KUKA KRL program: MyProgram_114().src

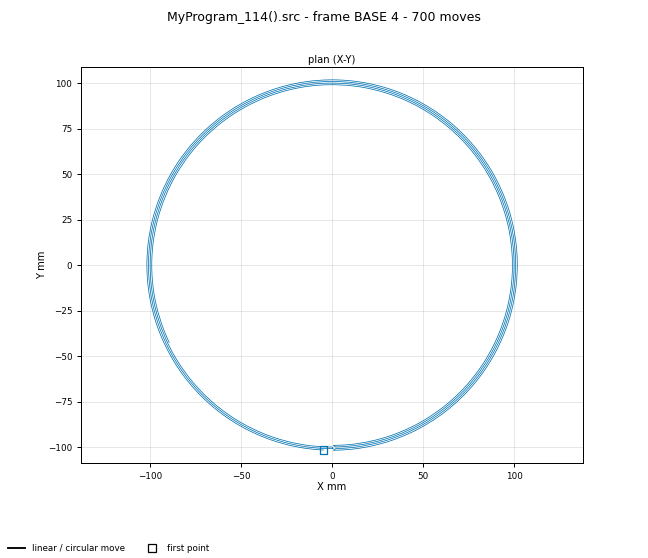
[picture p0: tool path of MyProgram_114().src in frame BASE 4, 700 of 700 moves have a stored position in this frame; points joined in program order, loops and branches not executed]
&ACCESS RVP
&REL 1
&PARAM TEMPLATE = C:\KRC\Roboter\Template\vorgabe
&PARAM EDITMASK = *
DEF MyProgram_114()
; ---- Setting reference (Base) ----
$BASE = BASE_DATA[4]

; --------------------------
; ---- Setting tool (TCP) ----
$TOOL = TOOL_DATA[3]
; --------------------------

$VEL.CP = VEL_APROX_PRINT
Startdeposition()
$VEL.CP = VEL_PRINT
LIN {X -4.7192,Y -101.6599,Z 99,A -97.1111,B 24.9445,C -1.7205,E1 24.9918,E2 182.675} C_DIS
LIN {X -7.4867,Y -101.4949,Z 99,A -98.6462,B 24.9445,C -1.7214,E1 24.9876,E2 184.2085} C_DIS
LIN {X -9.7017,Y -101.3059,Z 99,A -99.8982,B 24.9445,C -1.7214,E1 24.9841,E2 185.4609} C_DIS
LIN {X -12.4578,Y -101.0053,Z 99,A -101.4595,B 24.9445,C -1.7217,E1 24.9798,E2 187.0228} C_DIS
LIN {X -14.6609,Y -100.7078,Z 99,A -102.7373,B 24.9445,C -1.721,E1 24.9762,E2 188.3032} C_DIS
LIN {X -17.1279,Y -100.3177,Z 99,A -104.1189,B 24.9445,C -1.7223,E1 24.9724,E2 189.6829} C_DIS
LIN {X -19.8545,Y -99.8152,Z 99,A -105.6809,B 24.9444,C -1.7228,E1 24.9681,E2 191.2454} C_DIS
LIN {X -22.0297,Y -99.3564,Z 99,A -106.9595,B 24.9444,C -1.7224,E1 24.9646,E2 192.5265} C_DIS
LIN {X -24.4614,Y -98.7858,Z 99,A -108.3414,B 24.9443,C -1.7241,E1 24.9609,E2 193.9064} C_DIS
LIN {X -27.1435,Y -98.0841,Z 99,A -109.9045,B 24.9443,C -1.7249,E1 24.9567,E2 195.4699} C_DIS
LIN {X -29.2791,Y -97.4666,Z 99,A -111.184,B 24.9443,C -1.7248,E1 24.9532,E2 196.7519} C_DIS
LIN {X -31.5189,Y -96.7651,Z 99,A -112.5378,B 24.9443,C -1.7246,E1 24.9496,E2 198.1085} C_DIS
LIN {X -34.2855,Y -95.8216,Z 99,A -114.1306,B 24.944,C -1.7279,E1 24.9454,E2 199.6966} C_DIS
LIN {X -36.6268,Y -94.9513,Z 99,A -115.5395,B 24.944,C -1.7291,E1 24.9418,E2 201.1056} C_DIS
LIN {X -38.6915,Y -94.1274,Z 99,A -116.7915,B 24.9439,C -1.7303,E1 24.9385,E2 202.3574} C_DIS
LIN {X -40.9898,Y -93.1495,Z 99,A -118.2034,B 24.9439,C -1.7316,E1 24.9349,E2 203.7695} C_DIS
LIN {X -43.5126,Y -91.9996,Z 99,A -119.7683,B 24.9437,C -1.7333,E1 24.9309,E2 205.3344} C_DIS
LIN {X -45.5111,Y -91.026,Z 99,A -121.0488,B 24.9437,C -1.7338,E1 24.9277,E2 206.6171} C_DIS
LIN {X -48.4255,Y -89.509,Z 99,A -122.9613,B 24.9437,C -1.7339,E1 24.923,E2 208.5346} C_DIS
LIN {X -51.2454,Y -87.9271,Z 99,A -124.7043,B 24.9433,C -1.7392,E1 24.9188,E2 210.2701} C_DIS
LIN {X -53.1531,Y -86.7857,Z 99,A -125.9857,B 24.9433,C -1.74,E1 24.9157,E2 211.5535} C_DIS
LIN {X -55.4981,Y -85.3067,Z 99,A -127.5259,B 24.9431,C -1.7431,E1 24.9121,E2 213.0913} C_DIS
LIN {X -57.5749,Y -83.919,Z 99,A -128.9373,B 24.9429,C -1.7452,E1 24.9088,E2 214.5024} C_DIS
LIN {X -60.0996,Y -82.1274,Z 99,A -130.7649,B 24.9429,C -1.7452,E1 24.9047,E2 216.3365} C_DIS
LIN {X -62.3949,Y -80.3982,Z 99,A -132.3189,B 24.9426,C -1.7503,E1 24.9012,E2 217.8839} C_DIS
LIN {X -64.3492,Y -78.8428,Z 99,A -133.7487,B 24.9425,C -1.7521,E1 24.8981,E2 219.3149} C_DIS
LIN {X -66.4738,Y -77.0616,Z 99,A -135.2899,B 24.9422,C -1.7557,E1 24.8949,E2 220.8533} C_DIS
LIN {X -68.345,Y -75.4071,Z 99,A -136.7026,B 24.9421,C -1.7583,E1 24.8919,E2 222.2655} C_DIS
LIN {X -70.8764,Y -73.031,Z 99,A -138.666,B 24.9418,C -1.762,E1 24.8879,E2 224.2282} C_DIS
LIN {X -72.8404,Y -71.0742,Z 99,A -140.2343,B 24.9416,C -1.7651,E1 24.8849,E2 225.7959} C_DIS
LIN {X -74.5627,Y -69.2652,Z 99,A -141.6473,B 24.9414,C -1.7679,E1 24.8822,E2 227.2083} C_DIS
LIN {X -76.0569,Y -67.6192,Z 99,A -142.9199,B 24.9413,C -1.77,E1 24.8798,E2 228.4816} C_DIS
LIN {X -77.6934,Y -65.7323,Z 99,A -144.3182,B 24.941,C -1.7735,E1 24.8772,E2 229.8779} C_DIS
LIN {X -79.4561,Y -63.5924,Z 99,A -145.8873,B 24.9408,C -1.7769,E1 24.8745,E2 231.4463} C_DIS
LIN {X -80.9928,Y -61.6233,Z 99,A -147.3008,B 24.9406,C -1.78,E1 24.8721,E2 232.859} C_DIS
LIN {X -83.2061,Y -58.6004,Z 99,A -149.4215,B 24.9403,C -1.7848,E1 24.8686,E2 234.9785} C_DIS
LIN {X -85.1119,Y -55.7934,Z 99,A -151.3537,B 24.94,C -1.789,E1 24.8656,E2 236.9105} C_DIS
LIN {X -86.4974,Y -53.6208,Z 99,A -152.8276,B 24.9398,C -1.7919,E1 24.8634,E2 238.3848} C_DIS
LIN {X -87.9271,Y -51.2454,Z 99,A -154.3716,B 24.9395,C -1.7966,E1 24.8612,E2 239.9256} C_DIS
LIN {X -89.1582,Y -49.0722,Z 99,A -155.7862,B 24.9393,C -1.8002,E1 24.8593,E2 241.3392} C_DIS
LIN {X -90.2077,Y -47.1124,Z 99,A -157.0452,B 24.939,C -1.8033,E1 24.8576,E2 242.5974} C_DIS
LIN {X -91.4587,Y -44.6383,Z 99,A -158.6156,B 24.9388,C -1.8073,E1 24.8557,E2 244.1667} C_DIS
LIN {X -92.4107,Y -42.6294,Z 99,A -159.9009,B 24.9386,C -1.8097,E1 24.8542,E2 245.4533} C_DIS
LIN {X -93.5388,Y -40.0968,Z 99,A -161.4454,B 24.9383,C -1.8147,E1 24.8524,E2 246.9944} C_DIS
LIN {X -94.4947,Y -37.7892,Z 99,A -162.8609,B 24.938,C -1.8185,E1 24.8509,E2 248.4088} C_DIS
LIN {X -95.6293,Y -34.8126,Z 99,A -164.7206,B 24.9378,C -1.8215,E1 24.8491,E2 250.2717} C_DIS
LIN {X -96.5463,Y -32.1839,Z 99,A -166.2697,B 24.9374,C -1.8268,E1 24.8477,E2 251.817} C_DIS
LIN {X -97.3071,Y -29.8049,Z 99,A -167.6851,B 24.9372,C -1.8307,E1 24.8465,E2 253.2313} C_DIS
LIN {X -98.0787,Y -27.1626,Z 99,A -169.2166,B 24.9368,C -1.836,E1 24.8454,E2 254.759} C_DIS
LIN {X -98.7207,Y -24.7283,Z 99,A -170.6462,B 24.9365,C -1.8399,E1 24.8444,E2 256.1876} C_DIS
LIN {X -99.236,Y -22.5657,Z 99,A -171.932,B 24.9364,C -1.8426,E1 24.8436,E2 257.4745} C_DIS
LIN {X -99.7649,Y -20.0991,Z 99,A -173.3334,B 24.936,C -1.8477,E1 24.8428,E2 258.8721} C_DIS
LIN {X -100.1715,Y -17.9594,Z 99,A -174.6638,B 24.936,C -1.848,E1 24.8421,E2 260.2096} C_DIS
LIN {X -100.6272,Y -15.2044,Z 99,A -176.1799,B 24.9355,C -1.8548,E1 24.8414,E2 261.7185} C_DIS
LIN {X -100.97,Y -12.7303,Z 99,A -177.5957,B 24.9352,C -1.859,E1 24.8409,E2 263.1329} C_DIS
LIN {X -101.3347,Y -9.3895,Z 99,A -179.5206,B 24.9349,C -1.8639,E1 24.8404,E2 265.0576} C_DIS
LIN {X -101.5606,Y -6.5147,Z 99,A 178.89,B 24.9344,C -1.8702,E1 24.8401,E2 266.6414} C_DIS
LIN {X -101.7017,Y -3.7459,Z 99,A 177.3182,B 24.9341,C -1.8748,E1 24.8399,E2 268.2118} C_DIS
LIN {X -101.763,Y -1.2489,Z 99,A 175.8879,B 24.9338,C -1.8785,E1 24.8398,E2 269.6418} C_DIS
LIN {X -101.763,Y 1.2489,Z 99,A 174.2862,B 24.934,C -1.8764,E1 24.8398,E2 271.2582} C_DIS
LIN {X -101.6599,Y 4.7192,Z 99,A 172.4912,B 24.9332,C -1.8881,E1 24.84,E2 273.036} C_DIS
LIN {X -101.4949,Y 7.4867,Z 99,A 170.9451,B 24.9328,C -1.8936,E1 24.8403,E2 274.5783} C_DIS
LIN {X -101.3059,Y 9.7017,Z 99,A 169.6846,B 24.9325,C -1.8974,E1 24.8406,E2 275.8374} C_DIS
LIN {X -101.0053,Y 12.4578,Z 99,A 168.1128,B 24.9322,C -1.902,E1 24.8411,E2 277.4075} C_DIS
LIN {X -100.4783,Y 16.1671,Z 99,A 165.9887,B 24.9317,C -1.9083,E1 24.842,E2 279.5293} C_DIS
LIN {X -100.0513,Y 18.6281,Z 99,A 164.5726,B 24.9314,C -1.9125,E1 24.8427,E2 280.9438} C_DIS
LIN {X -99.6192,Y 20.8088,Z 99,A 163.2861,B 24.9312,C -1.9153,E1 24.8434,E2 282.2312} C_DIS
LIN {X -99.0786,Y 23.2473,Z 99,A 161.8959,B 24.9309,C -1.9203,E1 24.8443,E2 283.6176} C_DIS
LIN {X -98.4098,Y 25.9378,Z 99,A 160.3241,B 24.9305,C -1.9249,E1 24.8453,E2 285.1877} C_DIS
LIN {X -97.7436,Y 28.3451,Z 99,A 158.9084,B 24.9302,C -1.929,E1 24.8464,E2 286.6018} C_DIS
LIN {X -97.0186,Y 30.7353,Z 99,A 157.4927,B 24.9299,C -1.9331,E1 24.8476,E2 288.016} C_DIS
LIN {X -96.3229,Y 32.8467,Z 99,A 156.2321,B 24.9297,C -1.9367,E1 24.8487,E2 289.2751} C_DIS
LIN {X -95.5717,Y 34.9704,Z 99,A 154.8757,B 24.9297,C -1.9376,E1 24.85,E2 290.637} C_DIS
LIN {X -94.4947,Y 37.7892,Z 99,A 153.2451,B 24.9291,C -1.9451,E1 24.8516,E2 292.2587} C_DIS
LIN {X -93.6455,Y 39.8437,Z 99,A 151.9848,B 24.9288,C -1.9487,E1 24.853,E2 293.5177} C_DIS
LIN {X -92.6395,Y 42.1298,Z 99,A 150.5435,B 24.9286,C -1.9517,E1 24.8546,E2 294.9595} C_DIS
LIN {X -91.4587,Y 44.6383,Z 99,A 148.9981,B 24.9282,C -1.9569,E1 24.8565,E2 296.501} C_DIS
LIN {X -90.4607,Y 46.6247,Z 99,A 147.7128,B 24.928,C -1.9594,E1 24.8581,E2 297.7871} C_DIS
LIN {X -89.2892,Y 48.8307,Z 99,A 146.3231,B 24.9277,C -1.9641,E1 24.86,E2 299.173} C_DIS
LIN {X -87.9271,Y 51.2454,Z 99,A 144.6209,B 24.9277,C -1.9638,E1 24.8623,E2 300.8848} C_DIS
LIN {X -86.2717,Y 53.9822,Z 99,A 142.8532,B 24.9272,C -1.9701,E1 24.8649,E2 302.6466} C_DIS
LIN {X -84.7704,Y 56.3114,Z 99,A 141.3448,B 24.9268,C -1.9762,E1 24.8672,E2 304.148} C_DIS
LIN {X -83.363,Y 58.3748,Z 99,A 139.93,B 24.9265,C -1.9798,E1 24.8695,E2 305.5613} C_DIS
LIN {X -81.743,Y 60.6247,Z 99,A 138.3857,B 24.9262,C -1.9846,E1 24.872,E2 307.1017} C_DIS
LIN {X -80.2305,Y 62.6125,Z 99,A 136.9712,B 24.9259,C -1.988,E1 24.8744,E2 308.5145} C_DIS
LIN {X -78.8428,Y 64.3492,Z 99,A 135.7122,B 24.9257,C -1.9911,E1 24.8766,E2 309.7722} C_DIS
LIN {X -77.2398,Y 66.2647,Z 99,A 134.2982,B 24.9254,C -1.9945,E1 24.8792,E2 311.1846} C_DIS
LIN {X -75.4071,Y 68.345,Z 99,A 132.7287,B 24.9251,C -1.9981,E1 24.8821,E2 312.7524} C_DIS
LIN {X -73.7071,Y 70.175,Z 99,A 131.3148,B 24.9249,C -2.0013,E1 24.8848,E2 314.1649} C_DIS
LIN {X -71.9627,Y 71.9627,Z 99,A 129.901,B 24.9247,C -2.0045,E1 24.8875,E2 315.5771} C_DIS
LIN {X -70.175,Y 73.7071,Z 99,A 128.4875,B 24.9244,C -2.0076,E1 24.8904,E2 316.9892} C_DIS
LIN {X -68.5474,Y 75.2213,Z 99,A 127.2293,B 24.9242,C -2.0103,E1 24.893,E2 318.246} C_DIS
LIN {X -66.7956,Y 76.7806,Z 99,A 125.8457,B 24.9242,C -2.0111,E1 24.8959,E2 319.6332} C_DIS
LIN {X -64.7739,Y 78.4942,Z 99,A 124.3773,B 24.9239,C -2.0152,E1 24.899,E2 321.0975} C_DIS
LIN {X -62.8952,Y 80.0071,Z 99,A 122.9966,B 24.9237,C -2.0173,E1 24.902,E2 322.4781} C_DIS
LIN {X -60.6247,Y 81.743,Z 99,A 121.4223,B 24.9233,C -2.0219,E1 24.9055,E2 324.0472} C_DIS
LIN {X -58.6004,Y 83.2061,Z 99,A 120.0099,B 24.9231,C -2.0245,E1 24.9087,E2 325.4583} C_DIS
LIN {X -55.4981,Y 85.3067,Z 99,A 117.8912,B 24.9229,C -2.0283,E1 24.9137,E2 327.5749} C_DIS
LIN {X -53.6208,Y 86.4974,Z 99,A 116.6087,B 24.9228,C -2.0296,E1 24.9167,E2 328.8585} C_DIS
LIN {X -51.2454,Y 87.9271,Z 99,A 115.0673,B 24.9225,C -2.0331,E1 24.9204,E2 330.3962} C_DIS
LIN {X -49.312,Y 89.0243,Z 99,A 113.8175,B 24.9223,C -2.0353,E1 24.9234,E2 331.6443} C_DIS
LIN {X -47.1124,Y 90.2077,Z 99,A 112.3814,B 24.9223,C -2.0366,E1 24.927,E2 333.0813} C_DIS
LIN {X -44.6383,Y 91.4587,Z 99,A 110.8334,B 24.922,C -2.0396,E1 24.9308,E2 334.6264} C_DIS
LIN {X -42.3803,Y 92.5266,Z 99,A 109.4227,B 24.9218,C -2.0416,E1 24.9344,E2 336.0358} C_DIS
LIN {X -40.0968,Y 93.5388,Z 99,A 108.0119,B 24.9217,C -2.0435,E1 24.938,E2 337.4455} C_DIS
LIN {X -37.7892,Y 94.4947,Z 99,A 106.6008,B 24.9216,C -2.0453,E1 24.9417,E2 338.8555} C_DIS
LIN {X -35.7157,Y 95.2963,Z 99,A 105.3459,B 24.9214,C -2.0468,E1 24.9449,E2 340.1094} C_DIS
LIN {X -33.3663,Y 96.1441,Z 99,A 103.9356,B 24.9214,C -2.0485,E1 24.9486,E2 341.5186} C_DIS
LIN {X -30.7353,Y 97.0186,Z 99,A 102.371,B 24.9212,C -2.0502,E1 24.9528,E2 343.0819} C_DIS
LIN {X -27.7971,Y 97.8989,Z 99,A 100.5535,B 24.9212,C -2.0488,E1 24.9577,E2 344.9057} C_DIS
LIN {X -24.7283,Y 98.7207,Z 99,A 98.8471,B 24.9209,C -2.0535,E1 24.9623,E2 346.6034} C_DIS
LIN {X -21.2106,Y 99.5351,Z 99,A 96.8033,B 24.9209,C -2.055,E1 24.9678,E2 348.6464} C_DIS
LIN {X -18.8979,Y 99.9994,Z 99,A 95.4541,B 24.9208,C -2.0553,E1 24.9715,E2 349.9963} C_DIS
LIN {X -16.1671,Y 100.4783,Z 99,A 93.9164,B 24.9206,C -2.0572,E1 24.9757,E2 351.5309} C_DIS
LIN {X -12.7303,Y 100.97,Z 99,A 91.9591,B 24.9206,C -2.0584,E1 24.9812,E2 353.4869} C_DIS
LIN {X -9.9753,Y 101.2806,Z 99,A 90.3962,B 24.9205,C -2.0591,E1 24.9855,E2 355.0489} C_DIS
LIN {X -7.4867,Y 101.4949,Z 99,A 88.9887,B 24.9205,C -2.0597,E1 24.9894,E2 356.4557} C_DIS
LIN {X -5.2679,Y 101.6329,Z 99,A 87.7102,B 24.9205,C -2.0592,E1 24.993,E2 357.7357} C_DIS
LIN {X -1.6701,Y 101.7552,Z 99,A 85.685,B 24.9205,C -2.0599,E1 24.9986,E2 359.7597} C_DIS
LIN {X 1.2489,Y 101.763,Z 99,A 84.064,B 24.9203,C -2.061,E1 25.0032,E2 361.378} C_DIS
LIN {X 3.7459,Y 101.7017,Z 99,A 82.6575,B 24.9203,C -2.061,E1 25.0071,E2 362.7839} C_DIS
LIN {X 6.2407,Y 101.5791,Z 99,A 81.2508,B 24.9203,C -2.061,E1 25.011,E2 364.1901} C_DIS
LIN {X 9.332,Y 101.34,Z 99,A 79.429,B 24.9206,C -2.0582,E1 25.0161,E2 366.0178} C_DIS
LIN {X 12.4578,Y 101.0053,Z 99,A 77.7362,B 24.9204,C -2.0607,E1 25.0208,E2 367.7033} C_DIS
LIN {X 14.6609,Y 100.7078,Z 99,A 76.4597,B 24.9204,C -2.0595,E1 25.0243,E2 368.9817} C_DIS
LIN {X 17.1279,Y 100.3177,Z 99,A 75.08,B 24.9204,C -2.06,E1 25.0281,E2 370.3587} C_DIS
LIN {X 19.3148,Y 99.9191,Z 99,A 73.7784,B 24.9206,C -2.0576,E1 25.0317,E2 371.6645} C_DIS
LIN {X 22.0297,Y 99.3564,Z 99,A 72.3095,B 24.9204,C -2.0603,E1 25.0357,E2 373.125} C_DIS
LIN {X 24.4614,Y 98.7858,Z 99,A 70.8661,B 24.9206,C -2.0581,E1 25.0396,E2 374.5716} C_DIS
LIN {X 26.8783,Y 98.1558,Z 99,A 69.4615,B 24.9206,C -2.0573,E1 25.0434,E2 375.9759} C_DIS
LIN {X 28.9773,Y 97.5561,Z 99,A 68.1626,B 24.9209,C -2.0538,E1 25.0469,E2 377.281} C_DIS
LIN {X 31.6622,Y 96.7187,Z 99,A 66.628,B 24.9209,C -2.0544,E1 25.0509,E2 378.8114} C_DIS
LIN {X 34.8418,Y 95.6186,Z 99,A 64.6834,B 24.9211,C -2.0508,E1 25.0561,E2 380.7605} C_DIS
LIN {X 37.5335,Y 94.5951,Z 99,A 63.1452,B 24.9211,C -2.0524,E1 25.0601,E2 382.2916} C_DIS
LIN {X 40.0968,Y 93.5388,Z 99,A 61.5881,B 24.9211,C -2.0508,E1 25.0641,E2 383.8487} C_DIS
LIN {X 42.3803,Y 92.5266,Z 99,A 60.1853,B 24.9212,C -2.0493,E1 25.0676,E2 385.2515} C_DIS
LIN {X 44.3887,Y 91.5786,Z 99,A 58.9377,B 24.9214,C -2.048,E1 25.0708,E2 386.4992} C_DIS
LIN {X 46.6247,Y 90.4607,Z 99,A 57.509,B 24.9216,C -2.0453,E1 25.0744,E2 387.9301} C_DIS
LIN {X 49.0722,Y 89.1582,Z 99,A 55.9783,B 24.9216,C -2.0444,E1 25.0781,E2 389.4588} C_DIS
LIN {X 51.2454,Y 87.9271,Z 99,A 54.5765,B 24.9218,C -2.0425,E1 25.0815,E2 390.8607} C_DIS
LIN {X 53.1531,Y 86.7857,Z 99,A 53.3306,B 24.9218,C -2.0409,E1 25.0845,E2 392.1065} C_DIS
LIN {X 55.4981,Y 85.3067,Z 99,A 51.7733,B 24.9221,C -2.0386,E1 25.0881,E2 393.6643} C_DIS
LIN {X 57.3474,Y 84.073,Z 99,A 50.5259,B 24.9222,C -2.0367,E1 25.091,E2 394.9119} C_DIS
LIN {X 59.3934,Y 82.6403,Z 99,A 49.0996,B 24.9225,C -2.0335,E1 25.0943,E2 396.3408} C_DIS
LIN {X 61.6233,Y 80.9928,Z 99,A 47.57,B 24.9225,C -2.0319,E1 25.0977,E2 397.8686} C_DIS
LIN {X 63.3768,Y 79.6265,Z 99,A 46.3236,B 24.9227,C -2.0299,E1 25.1004,E2 399.1152} C_DIS
LIN {X 65.5132,Y 77.8799,Z 99,A 44.7761,B 24.9229,C -2.0271,E1 25.1038,E2 400.6632} C_DIS
LIN {X 67.4145,Y 76.2401,Z 99,A 43.3691,B 24.9231,C -2.0246,E1 25.1067,E2 402.0707} C_DIS
LIN {X 69.2652,Y 74.5627,Z 99,A 41.9687,B 24.9233,C -2.022,E1 25.1096,E2 403.4716} C_DIS
LIN {X 70.8764,Y 73.031,Z 99,A 40.7229,B 24.9235,C -2.0196,E1 25.1121,E2 404.7179} C_DIS
LIN {X 73.031,Y 70.8764,Z 99,A 38.891,B 24.9241,C -2.0113,E1 25.1157,E2 406.5616} C_DIS
LIN {X 75.4071,Y 68.345,Z 99,A 37.07,B 24.9241,C -2.0123,E1 25.1192,E2 408.3724} C_DIS
LIN {X 76.9394,Y 66.6138,Z 99,A 35.7823,B 24.9243,C -2.0098,E1 25.1215,E2 409.66} C_DIS
LIN {X 78.4942,Y 64.7739,Z 99,A 34.4255,B 24.9245,C -2.0066,E1 25.124,E2 411.0181} C_DIS
LIN {X 80.0602,Y 62.8281,Z 99,A 33.0266,B 24.9247,C -2.0036,E1 25.1264,E2 412.4178} C_DIS
LIN {X 81.3585,Y 61.1365,Z 99,A 31.7578,B 24.9252,C -1.9979,E1 25.1286,E2 413.6938} C_DIS
LIN {X 83.0466,Y 58.824,Z 99,A 30.2036,B 24.9252,C -1.9962,E1 25.1311,E2 415.2446} C_DIS
LIN {X 84.6192,Y 56.5407,Z 99,A 28.6769,B 24.9255,C -1.9936,E1 25.1335,E2 416.7699} C_DIS
LIN {X 85.8329,Y 54.6783,Z 99,A 27.4324,B 24.9257,C -1.9906,E1 25.1354,E2 418.0152} C_DIS
LIN {X 87.2916,Y 52.3206,Z 99,A 25.8803,B 24.926,C -1.9868,E1 25.1376,E2 419.5683} C_DIS
LIN {X 88.5493,Y 50.1626,Z 99,A 24.4823,B 24.9262,C -1.9834,E1 25.1396,E2 420.9672} C_DIS
LIN {X 89.7537,Y 47.9744,Z 99,A 23.0843,B 24.9265,C -1.9798,E1 25.1414,E2 422.3662} C_DIS
LIN {X 90.904,Y 45.7572,Z 99,A 21.6867,B 24.9268,C -1.9763,E1 25.1432,E2 423.7647} C_DIS
LIN {X 91.8806,Y 43.7602,Z 99,A 20.4428,B 24.927,C -1.9731,E1 25.1447,E2 425.0096} C_DIS
LIN {X 93.0397,Y 41.2417,Z 99,A 18.8915,B 24.9273,C -1.969,E1 25.1465,E2 426.5621} C_DIS
LIN {X 93.9171,Y 39.1991,Z 99,A 17.6475,B 24.9276,C -1.9657,E1 25.1479,E2 427.8069} C_DIS
LIN {X 94.8509,Y 36.8825,Z 99,A 16.2503,B 24.9278,C -1.962,E1 25.1493,E2 429.2053} C_DIS
LIN {X 95.8216,Y 34.2855,Z 99,A 14.6991,B 24.9281,C -1.9577,E1 25.1508,E2 430.7578} C_DIS
LIN {X 96.5463,Y 32.1839,Z 99,A 13.4386,B 24.9284,C -1.9537,E1 25.1519,E2 432.0208} C_DIS
LIN {X 97.3071,Y 29.8049,Z 99,A 12.0586,B 24.9287,C -1.9505,E1 25.1531,E2 433.4005} C_DIS
LIN {X 98.0092,Y 27.4078,Z 99,A 10.641,B 24.929,C -1.9458,E1 25.1542,E2 434.8211} C_DIS
LIN {X 98.6523,Y 24.9943,Z 99,A 9.2649,B 24.9292,C -1.9427,E1 25.1551,E2 436.1966} C_DIS
LIN {X 99.2978,Y 22.2981,Z 99,A 7.7145,B 24.9296,C -1.9382,E1 25.1561,E2 437.7484} C_DIS
LIN {X 100.0513,Y 18.6281,Z 99,A 5.6193,B 24.93,C -1.9322,E1 25.1573,E2 439.8456} C_DIS
LIN {X 100.4783,Y 16.1671,Z 99,A 4.2228,B 24.9303,C -1.9282,E1 25.1579,E2 441.2434} C_DIS
LIN {X 100.8062,Y 13.9684,Z 99,A 2.9542,B 24.9306,C -1.9236,E1 25.1584,E2 442.5154} C_DIS
LIN {X 101.2337,Y 10.4231,Z 99,A 0.9391,B 24.9311,C -1.917,E1 25.1591,E2 444.5341} C_DIS
LIN {X 101.473,Y 7.7606,Z 99,A -0.5119,B 24.9313,C -1.9144,E1 25.1594,E2 445.9826} C_DIS
LIN {X 101.6329,Y 5.2679,Z 99,A -1.9339,B 24.9317,C -1.9092,E1 25.1596,E2 447.4084} C_DIS
LIN {X 101.7316,Y 2.7722,Z 99,A -3.3304,B 24.932,C -1.9051,E1 25.1597,E2 448.8063} C_DIS
LIN {X 101.7703,Y 0,Z 99,A -4.8381,B 24.9322,C -1.9022,E1 25.1597,E2 450.3118} C_DIS
LIN {X 101.7163,Y -3.2698,Z 99,A -6.7172,B 24.9327,C -1.8948,E1 25.1597,E2 452.1973} C_DIS
LIN {X 101.5791,Y -6.2407,Z 99,A -8.3461,B 24.933,C -1.8912,E1 25.1594,E2 453.825} C_DIS
LIN {X 101.4173,Y -8.4578,Z 99,A -9.5887,B 24.9332,C -1.8875,E1 25.1592,E2 455.0689} C_DIS
LIN {X 101.1848,Y -10.8905,Z 99,A -10.98,B 24.9336,C -1.8825,E1 25.1588,E2 456.4638} C_DIS
LIN {X 100.8448,Y -13.6964,Z 99,A -12.535,B 24.9338,C -1.8788,E1 25.1582,E2 458.0184} C_DIS
LIN {X 100.4783,Y -16.1671,Z 99,A -13.9314,B 24.9341,C -1.8747,E1 25.1576,E2 459.4163} C_DIS
LIN {X 100.0999,Y -18.3577,Z 99,A -15.2001,B 24.9345,C -1.87,E1 25.157,E2 460.6887} C_DIS
LIN {X 99.6192,Y -20.8088,Z 99,A -16.571,B 24.9347,C -1.8669,E1 25.1562,E2 462.0588} C_DIS
LIN {X 99.0167,Y -23.5149,Z 99,A -18.1213,B 24.935,C -1.8623,E1 25.1553,E2 463.6109} C_DIS
LIN {X 98.1869,Y -26.7629,Z 99,A -20.0133,B 24.9354,C -1.8562,E1 25.1539,E2 465.5065} C_DIS
LIN {X 97.4666,Y -29.2791,Z 99,A -21.4848,B 24.9357,C -1.8516,E1 25.1528,E2 466.9804} C_DIS
LIN {X 96.7187,Y -31.6622,Z 99,A -22.8814,B 24.936,C -1.8476,E1 25.1516,E2 468.3785} C_DIS
LIN {X 95.8216,Y -34.2855,Z 99,A -24.4063,B 24.9363,C -1.8441,E1 25.1502,E2 469.903} C_DIS
LIN {X 94.9513,Y -36.6268,Z 99,A -25.803,B 24.9365,C -1.8402,E1 25.1488,E2 471.3012} C_DIS
LIN {X 94.1274,Y -38.6915,Z 99,A -27.0719,B 24.9368,C -1.8357,E1 25.1475,E2 472.5738} C_DIS
LIN {X 93.1495,Y -40.9898,Z 99,A -28.4432,B 24.937,C -1.8328,E1 25.1459,E2 473.9444} C_DIS
LIN {X 91.9996,Y -43.5126,Z 99,A -29.9941,B 24.9373,C -1.8285,E1 25.1441,E2 475.497} C_DIS
LIN {X 91.026,Y -45.5111,Z 99,A -31.2628,B 24.9376,C -1.824,E1 25.1425,E2 476.7695} C_DIS
LIN {X 89.7537,Y -47.9744,Z 99,A -32.7885,B 24.9379,C -1.8208,E1 25.1406,E2 478.2946} C_DIS
LIN {X 88.6833,Y -49.9227,Z 99,A -34.0575,B 24.9382,C -1.8165,E1 25.1388,E2 479.5673} C_DIS
LIN {X 87.4314,Y -52.0841,Z 99,A -35.4293,B 24.9383,C -1.8138,E1 25.1369,E2 480.9384} C_DIS
LIN {X 85.9813,Y -54.4471,Z 99,A -36.9806,B 24.9386,C -1.8097,E1 25.1346,E2 482.4914} C_DIS
LIN {X 84.7704,Y -56.3114,Z 99,A -38.2473,B 24.9389,C -1.8056,E1 25.1327,E2 483.7615} C_DIS
LIN {X 83.2061,Y -58.6004,Z 99,A -39.7761,B 24.9391,C -1.8025,E1 25.1302,E2 485.2901} C_DIS
LIN {X 81.7472,Y -60.6189,Z 99,A -41.1691,B 24.9393,C -1.7991,E1 25.1279,E2 486.6845} C_DIS
LIN {X 80.3982,Y -62.3949,Z 99,A -42.4439,B 24.9396,C -1.7949,E1 25.1257,E2 487.963} C_DIS
LIN {X 78.8428,Y -64.3492,Z 99,A -43.8423,B 24.9398,C -1.7915,E1 25.1233,E2 489.363} C_DIS
LIN {X 77.0616,Y -66.4738,Z 99,A -45.3684,B 24.94,C -1.7888,E1 25.1205,E2 490.8884} C_DIS
LIN {X 75.4071,Y -68.345,Z 99,A -46.7672,B 24.9402,C -1.7855,E1 25.1179,E2 492.2888} C_DIS
LIN {X 73.8953,Y -69.9749,Z 99,A -48.012,B 24.9404,C -1.7827,E1 25.1155,E2 493.5349} C_DIS
LIN {X 72.1558,Y -71.7673,Z 99,A -49.4362,B 24.9407,C -1.7785,E1 25.1128,E2 494.9629} C_DIS
LIN {X 70.175,Y -73.7071,Z 99,A -50.9634,B 24.9409,C -1.7761,E1 25.1097,E2 496.4895} C_DIS
LIN {X 68.5744,Y -75.1966,Z 99,A -52.1928,B 24.9411,C -1.7733,E1 25.1072,E2 497.7205} C_DIS
LIN {X 66.4738,Y -77.0616,Z 99,A -53.7618,B 24.9413,C -1.7701,E1 25.1039,E2 499.2908} C_DIS
LIN {X 64.7739,Y -78.4942,Z 99,A -55.0329,B 24.9415,C -1.7665,E1 25.1011,E2 500.5654} C_DIS
LIN {X 62.8281,Y -80.0602,Z 99,A -56.4324,B 24.9417,C -1.7637,E1 25.0981,E2 501.9663} C_DIS
LIN {X 60.6247,Y -81.743,Z 99,A -57.9605,B 24.9418,C -1.7617,E1 25.0947,E2 503.4937} C_DIS
LIN {X 58.6004,Y -83.2061,Z 99,A -59.3604,B 24.942,C -1.7591,E1 25.0915,E2 504.895} C_DIS
LIN {X 56.7682,Y -84.4652,Z 99,A -60.6323,B 24.9422,C -1.7558,E1 25.0885,E2 506.1704} C_DIS
LIN {X 54.6783,Y -85.8329,Z 99,A -62.007,B 24.9423,C -1.7543,E1 25.0853,E2 507.544} C_DIS
LIN {X 52.3206,Y -87.2916,Z 99,A -63.5616,B 24.9425,C -1.7516,E1 25.0816,E2 509.1001} C_DIS
LIN {X 50.4008,Y -88.4125,Z 99,A -64.834,B 24.9427,C -1.7485,E1 25.0785,E2 510.376} C_DIS
LIN {X 48.2158,Y -89.6227,Z 99,A -66.2092,B 24.9427,C -1.7473,E1 25.0751,E2 511.7501} C_DIS
LIN {X 46.0019,Y -90.779,Z 99,A -67.636,B 24.943,C -1.7441,E1 25.0716,E2 513.1804} C_DIS
LIN {X 43.7602,Y -91.8806,Z 99,A -69.0117,B 24.943,C -1.743,E1 25.0681,E2 514.555} C_DIS
LIN {X 41.2417,Y -93.0397,Z 99,A -70.5676,B 24.9432,C -1.7408,E1 25.0642,E2 516.1124} C_DIS
LIN {X 39.1991,Y -93.9171,Z 99,A -71.8406,B 24.9434,C -1.7382,E1 25.0609,E2 517.3887} C_DIS
LIN {X 36.6268,Y -94.9513,Z 99,A -73.3712,B 24.9434,C -1.7371,E1 25.0569,E2 518.9183} C_DIS
LIN {X 34.5436,Y -95.7274,Z 99,A -74.6192,B 24.9435,C -1.7356,E1 25.0536,E2 520.1672} C_DIS
LIN {X 32.1839,Y -96.5463,Z 99,A -76.0473,B 24.9437,C -1.733,E1 25.0499,E2 521.5987} C_DIS
LIN {X 29.8049,Y -97.3071,Z 99,A -77.4498,B 24.9438,C -1.7315,E1 25.0461,E2 523.0023} C_DIS
LIN {X 26.2031,Y -98.3382,Z 99,A -79.5408,B 24.9439,C -1.7299,E1 25.0405,E2 525.0936} C_DIS
LIN {X 23.5149,Y -99.0167,Z 99,A -81.086,B 24.9439,C -1.7289,E1 25.0363,E2 526.6388} C_DIS
LIN {X 21.0779,Y -99.564,Z 99,A -82.4896,B 24.9441,C -1.7277,E1 25.0325,E2 528.0434} C_DIS
LIN {X 17.8047,Y -100.1994,Z 99,A -84.4163,B 24.9443,C -1.7243,E1 25.0272,E2 529.976} C_DIS
LIN {X 15.2044,Y -100.6272,Z 99,A -85.8705,B 24.9443,C -1.7243,E1 25.0232,E2 531.4287} C_DIS
LIN {X 12.7303,Y -100.97,Z 99,A -87.2489,B 24.9443,C -1.7245,E1 25.0194,E2 532.8056} C_DIS
LIN {X 9.9753,Y -101.2806,Z 99,A -88.808,B 24.9443,C -1.7237,E1 25.015,E2 534.3656} C_DIS
LIN {X 7.4867,Y -101.4949,Z 99,A -90.2126,B 24.9443,C -1.723,E1 25.0111,E2 535.771} C_DIS
LIN {X 5.268,Y -101.6329,Z 99,A -91.4889,B 24.9445,C -1.7216,E1 25.0075,E2 537.0502} C_DIS
LIN {X 2.7722,Y -101.7316,Z 99,A -92.8942,B 24.9445,C -1.7212,E1 25.0036,E2 538.4562} C_DIS
LIN {X 0.7009,Y -101.7664,Z 99,A -93.7509,B 24.9437,C -1.7327,E1 25.0013,E2 539.2856} C_DIS
Enddeposition()
LIN {X 0.7009,Y -101.7664,Z 99,A -93.7509,B 24.9437,C -1.7327,E1 25.0013,E2 539.2856} C_DIS
Startdeposition()
$VEL.CP = VEL_PRINT
LIN {X 2.0126,Y -100.8623,Z 99,A -92.6029,B 24.9417,C -1.7637,E1 25.0047,E2 538.0642} C_DIS
LIN {X 6.1987,Y -100.6934,Z 99,A -90.1204,B 24.9414,C -1.7685,E1 25.0117,E2 535.571} C_DIS
LIN {X 9.309,Y -100.4518,Z 99,A -88.4765,B 24.9416,C -1.7645,E1 25.0162,E2 533.9375} C_DIS
LIN {X 12.6601,Y -100.0852,Z 99,A -86.0935,B 24.9404,C -1.7839,E1 25.0229,E2 531.5105} C_DIS
LIN {X 15.9238,Y -99.6189,Z 99,A -84.565,B 24.9412,C -1.7718,E1 25.0271,E2 530.012} C_DIS
LIN {X 23.7631,Y -98.0437,Z 99,A -80.1805,B 24.9413,C -1.7697,E1 25.039,E2 525.6381} C_DIS
LIN {X 28.9508,Y -96.6393,Z 99,A -77.1387,B 24.9411,C -1.7726,E1 25.0472,E2 522.5944} C_DIS
LIN {X 32.2678,Y -95.5825,Z 99,A -75.0278,B 24.9406,C -1.7802,E1 25.0528,E2 520.4694} C_DIS
LIN {X 38.5515,Y -93.2272,Z 99,A -71.1936,B 24.9402,C -1.7863,E1 25.0629,E2 516.6292} C_DIS
LIN {X 42.0759,Y -91.6905,Z 99,A -69.0703,B 24.9402,C -1.7873,E1 25.0683,E2 514.5089} C_DIS
LIN {X 45.9589,Y -89.8054,Z 99,A -66.8041,B 24.9404,C -1.784,E1 25.0739,E2 512.2567} C_DIS
LIN {X 48.5707,Y -88.4217,Z 99,A -64.861,B 24.9394,C -1.7974,E1 25.0787,E2 510.2874} C_DIS
LIN {X 52.065,Y -86.4095,Z 99,A -62.8289,B 24.9399,C -1.7913,E1 25.0836,E2 508.2759} C_DIS
LIN {X 53.9523,Y -85.2451,Z 99,A -61.3231,B 24.939,C -1.8035,E1 25.0872,E2 506.7461} C_DIS
LIN {X 56.477,Y -83.5917,Z 99,A -59.7209,B 24.9391,C -1.8025,E1 25.0909,E2 505.1517} C_DIS
LIN {X 59.8226,Y -81.2315,Z 99,A -57.3608,B 24.9387,C -1.8087,E1 25.0962,E2 502.7852} C_DIS
LIN {X 62.4073,Y -79.2628,Z 99,A -55.6186,B 24.9387,C -1.8085,E1 25.1001,E2 501.0498} C_DIS
LIN {X 64.9092,Y -77.2291,Z 99,A -53.6084,B 24.9379,C -1.8198,E1 25.1044,E2 499.0207} C_DIS
LIN {X 68.0745,Y -74.4521,Z 99,A -51.3043,B 24.9378,C -1.8218,E1 25.1092,E2 496.7209} C_DIS
LIN {X 70.5601,Y -72.1021,Z 99,A -49.5352,B 24.938,C -1.8194,E1 25.1128,E2 494.9647} C_DIS
LIN {X 72.7507,Y -69.8898,Z 99,A -47.7901,B 24.9377,C -1.8229,E1 25.1162,E2 493.219} C_DIS
LIN {X 75.0312,Y -67.4358,Z 99,A -45.7887,B 24.9371,C -1.8317,E1 25.12,E2 491.2056} C_DIS
LIN {X 77.4663,Y -64.6238,Z 99,A -43.7986,B 24.9371,C -1.8322,E1 25.1235,E2 489.2233} C_DIS
LIN {X 79.3388,Y -62.3111,Z 99,A -42.1053,B 24.9368,C -1.8369,E1 25.1265,E2 487.5271} C_DIS
LIN {X 81.2834,Y -59.7518,Z 99,A -40.5065,B 24.937,C -1.8326,E1 25.1292,E2 485.946} C_DIS
LIN {X 82.7202,Y -57.7464,Z 99,A -38.7967,B 24.9359,C -1.849,E1 25.132,E2 484.2057} C_DIS
LIN {X 84.8219,Y -54.6121,Z 99,A -36.9041,B 24.9362,C -1.8448,E1 25.1348,E2 482.3324} C_DIS
LIN {X 86.3817,Y -52.1108,Z 99,A -35.0641,B 24.9354,C -1.8564,E1 25.1376,E2 480.4745} C_DIS
LIN {X 88.8341,Y -47.8103,Z 99,A -31.4317,B 24.9324,C -1.8985,E1 25.1426,E2 476.7618} C_DIS
LIN {X 90.9838,Y -43.5796,Z 99,A -29.1179,B 24.933,C -1.8907,E1 25.1453,E2 474.4786} C_DIS
LIN {X 92.3876,Y -40.5192,Z 99,A -27.6784,B 24.934,C -1.8771,E1 25.1469,E2 473.0793} C_DIS
LIN {X 93.4963,Y -37.8906,Z 99,A -26.0088,B 24.9335,C -1.8841,E1 25.1487,E2 471.4024} C_DIS
LIN {X 94.793,Y -34.5183,Z 99,A -24.0805,B 24.9334,C -1.8853,E1 25.1506,E2 469.4818} C_DIS
LIN {X 96.3822,Y -29.7944,Z 99,A -20.554,B 24.9307,C -1.923,E1 25.1536,E2 465.8865} C_DIS
LIN {X 97.5405,Y -25.7549,Z 99,A -18.9777,B 24.9325,C -1.897,E1 25.1548,E2 464.3805} C_DIS
LIN {X 98.3123,Y -22.6258,Z 99,A -16.8621,B 24.9313,C -1.9146,E1 25.1561,E2 462.2358} C_DIS
LIN {X 99.0996,Y -18.8823,Z 99,A -14.3721,B 24.9298,C -1.9347,E1 25.1575,E2 459.7129} C_DIS
LIN {X 99.695,Y -15.4315,Z 99,A -12.8951,B 24.9309,C -1.9199,E1 25.1581,E2 458.2794} C_DIS
LIN {X 100.2307,Y -11.4508,Z 99,A -10.4325,B 24.9298,C -1.9347,E1 25.159,E2 455.7963} C_DIS
LIN {X 100.5789,Y -7.8207,Z 99,A -8.5851,B 24.93,C -1.9322,E1 25.1594,E2 453.9659} C_DIS
LIN {X 100.8002,Y -4.0755,Z 99,A -6.3529,B 24.9292,C -1.9433,E1 25.1597,E2 451.7209} C_DIS
LIN {X 100.8803,Y -0.6215,Z 99,A -4.6987,B 24.9297,C -1.937,E1 25.1597,E2 450.0914} C_DIS
LIN {X 100.8606,Y 2.1017,Z 99,A -2.9846,B 24.9288,C -1.9488,E1 25.1597,E2 448.3595} C_DIS
LIN {X 100.7847,Y 4.4361,Z 99,A -1.2942,B 24.9274,C -1.968,E1 25.1595,E2 446.6338} C_DIS
LIN {X 100.4359,Y 9.482,Z 99,A 1.2089,B 24.9278,C -1.962,E1 25.1589,E2 444.1598} C_DIS
LIN {X 99.8806,Y 14.1806,Z 99,A 4.2067,B 24.9262,C -1.9833,E1 25.1579,E2 441.1294} C_DIS
LIN {X 98.768,Y 20.547,Z 99,A 8.7001,B 24.9228,C -2.0288,E1 25.1554,E2 436.5548} C_DIS
LIN {X 97.3265,Y 26.549,Z 99,A 11.0153,B 24.9257,C -1.9904,E1 25.1538,E2 434.3437} C_DIS
LIN {X 96.4353,Y 29.6233,Z 99,A 12.6887,B 24.9257,C -1.99,E1 25.1525,E2 432.6808} C_DIS
LIN {X 95.4355,Y 32.7037,Z 99,A 14.7546,B 24.9246,C -2.0047,E1 25.1506,E2 430.5918} C_DIS
LIN {X 94.1737,Y 36.177,Z 99,A 16.8064,B 24.9243,C -2.009,E1 25.1486,E2 428.5414} C_DIS
LIN {X 92.7954,Y 39.5782,Z 99,A 19.9076,B 24.9207,C -2.0567,E1 25.1451,E2 425.3445} C_DIS
LIN {X 90.328,Y 44.9232,Z 99,A 22.0616,B 24.9237,C -2.0174,E1 25.1426,E2 423.2948} C_DIS
LIN {X 88.7162,Y 48.0278,Z 99,A 23.9991,B 24.9234,C -2.0209,E1 25.1401,E2 421.3594} C_DIS
LIN {X 87.5748,Y 50.0793,Z 99,A 25.4607,B 24.9228,C -2.0297,E1 25.1381,E2 419.8846} C_DIS
LIN {X 85.8311,Y 53.0142,Z 99,A 27.4187,B 24.9223,C -2.0355,E1 25.1352,E2 417.9227} C_DIS
LIN {X 83.8965,Y 56.0263,Z 99,A 29.5198,B 24.9217,C -2.0435,E1 25.132,E2 415.8133} C_DIS
LIN {X 81.582,Y 59.3439,Z 99,A 31.6631,B 24.9217,C -2.0431,E1 25.1285,E2 413.6814} C_DIS
LIN {X 79.5024,Y 62.1041,Z 99,A 33.7078,B 24.9211,C -2.0511,E1 25.125,E2 411.6274} C_DIS
LIN {X 77.0644,Y 65.1037,Z 99,A 35.6587,B 24.9215,C -2.0465,E1 25.1216,E2 409.6963} C_DIS
LIN {X 74.0646,Y 68.4966,Z 99,A 38.4293,B 24.9204,C -2.0603,E1 25.1164,E2 406.9057} C_DIS
LIN {X 71.7537,Y 70.9129,Z 99,A 40.2395,B 24.9204,C -2.0608,E1 25.1129,E2 405.1018} C_DIS
LIN {X 68.5776,Y 73.9905,Z 99,A 42.8395,B 24.9197,C -2.0695,E1 25.1076,E2 402.492} C_DIS
LIN {X 65.8305,Y 76.4451,Z 99,A 44.7312,B 24.92,C -2.0657,E1 25.1037,E2 400.6168} C_DIS
LIN {X 63.9348,Y 78.0375,Z 99,A 46.3153,B 24.9192,C -2.0754,E1 25.1002,E2 399.0158} C_DIS
LIN {X 61.0825,Y 80.2901,Z 99,A 48.1728,B 24.9196,C -2.071,E1 25.0962,E2 397.1756} C_DIS
LIN {X 58.7133,Y 82.0366,Z 99,A 49.9778,B 24.9189,C -2.0792,E1 25.0921,E2 395.3577} C_DIS
LIN {X 55.6807,Y 84.1244,Z 99,A 52.0648,B 24.9187,C -2.0824,E1 25.0872,E2 393.27} C_DIS
LIN {X 52.5575,Y 86.1102,Z 99,A 54.0803,B 24.9187,C -2.0823,E1 25.0825,E2 391.2613} C_DIS
LIN {X 48.2597,Y 88.5904,Z 99,A 57.3555,B 24.917,C -2.1041,E1 25.0744,E2 387.9442} C_DIS
LIN {X 45.3366,Y 90.1225,Z 99,A 58.8413,B 24.918,C -2.0913,E1 25.0708,E2 386.4927} C_DIS
LIN {X 42.0569,Y 91.6993,Z 99,A 60.9082,B 24.9178,C -2.0938,E1 25.0655,E2 384.4252} C_DIS
LIN {X 39.4462,Y 92.851,Z 99,A 62.5238,B 24.9177,C -2.0954,E1 25.0614,E2 382.8098} C_DIS
LIN {X 36.0138,Y 94.2355,Z 99,A 64.5587,B 24.9177,C -2.0949,E1 25.0561,E2 380.7806} C_DIS
LIN {X 33.2882,Y 95.232,Z 99,A 66.2931,B 24.9173,C -2.0997,E1 25.0515,E2 379.0383} C_DIS
LIN {X 29.4675,Y 96.4836,Z 99,A 68.6038,B 24.9171,C -2.1025,E1 25.0454,E2 376.7252} C_DIS
LIN {X 23.7377,Y 98.0499,Z 99,A 72.5964,B 24.9151,C -2.1282,E1 25.0344,E2 372.6776} C_DIS
LIN {X 19.4273,Y 98.9946,Z 99,A 74.192,B 24.9177,C -2.0947,E1 25.0303,E2 371.1635} C_DIS
LIN {X 15.8177,Y 99.6353,Z 99,A 76.4486,B 24.9171,C -2.102,E1 25.0241,E2 368.892} C_DIS
LIN {X 13.361,Y 99.9944,Z 99,A 77.9665,B 24.9168,C -2.1064,E1 25.0198,E2 367.3649} C_DIS
LIN {X 9.4688,Y 100.4371,Z 99,A 80.08,B 24.9171,C -2.1025,E1 25.014,E2 365.2619} C_DIS
LIN {X 4.4556,Y 100.7839,Z 99,A 82.912,B 24.9171,C -2.1017,E1 25.0061,E2 362.433} C_DIS
LIN {X 2.0889,Y 100.8609,Z 99,A 84.3654,B 24.9169,C -2.1056,E1 25.002,E2 360.9707} C_DIS
LIN {X -1.654,Y 100.8689,Z 99,A 86.4296,B 24.9171,C -2.1028,E1 24.9963,E2 358.9131} C_DIS
LIN {X -4.9537,Y 100.7624,Z 99,A 88.5211,B 24.9165,C -2.1102,E1 24.9904,E2 356.8037} C_DIS
LIN {X -9.9425,Y 100.3927,Z 99,A 91.8234,B 24.9152,C -2.1259,E1 24.9811,E2 353.4623} C_DIS
LIN {X -14.076,Y 99.8955,Z 99,A 93.3492,B 24.9178,C -2.0936,E1 24.9771,E2 352.0122} C_DIS
LIN {X -21.4511,Y 98.5752,Z 99,A 97.8493,B 24.9174,C -2.0991,E1 24.9647,E2 347.4943} C_DIS
LIN {X -24.6332,Y 97.8298,Z 99,A 99.5045,B 24.9181,C -2.09,E1 24.9602,E2 345.8584} C_DIS
LIN {X -27.4401,Y 97.0787,Z 99,A 101.0292,B 24.9186,C -2.0837,E1 24.9562,E2 344.3461} C_DIS
LIN {X -30.0398,Y 96.3061,Z 99,A 102.8349,B 24.918,C -2.0916,E1 24.9513,E2 342.5188} C_DIS
LIN {X -32.9009,Y 95.3679,Z 99,A 104.6306,B 24.9179,C -2.0926,E1 24.9465,E2 340.7173} C_DIS
LIN {X -36.4505,Y 94.0681,Z 99,A 106.7677,B 24.9181,C -2.0894,E1 24.9409,E2 338.5833} C_DIS
LIN {X -39.9318,Y 92.6437,Z 99,A 108.9509,B 24.9182,C -2.088,E1 24.9353,E2 336.3983} C_DIS
LIN {X -42.9107,Y 91.3019,Z 99,A 110.7757,B 24.9185,C -2.0841,E1 24.9307,E2 334.5784} C_DIS
LIN {X -45.7713,Y 89.9013,Z 99,A 112.3386,B 24.9195,C -2.0724,E1 24.9269,E2 333.039} C_DIS
LIN {X -49.7629,Y 87.7565,Z 99,A 115.1937,B 24.919,C -2.078,E1 24.9198,E2 330.1626} C_DIS
LIN {X -52.9485,Y 85.8722,Z 99,A 117.2866,B 24.9194,C -2.0738,E1 24.9148,E2 328.0733} C_DIS
LIN {X -55.8804,Y 83.9927,Z 99,A 119.3268,B 24.9194,C -2.0722,E1 24.9101,E2 326.0302} C_DIS
LIN {X -58.7636,Y 82.0007,Z 99,A 121.2844,B 24.9199,C -2.067,E1 24.9056,E2 324.0782} C_DIS
LIN {X -61.7238,Y 79.7962,Z 99,A 123.3611,B 24.9203,C -2.0619,E1 24.901,E2 322.0061} C_DIS
LIN {X -64.1125,Y 77.8912,Z 99,A 125.1681,B 24.9203,C -2.0606,E1 24.8971,E2 320.1954} C_DIS
LIN {X -67.1123,Y 75.3208,Z 99,A 127.2419,B 24.9212,C -2.0496,E1 24.8927,E2 318.1396} C_DIS
LIN {X -68.8613,Y 73.7257,Z 99,A 128.7057,B 24.9212,C -2.0507,E1 24.8897,E2 316.6674} C_DIS
LIN {X -71.5439,Y 71.1253,Z 99,A 130.6672,B 24.922,C -2.04,E1 24.8859,E2 314.7231} C_DIS
LIN {X -73.7768,Y 68.8069,Z 99,A 132.6645,B 24.9219,C -2.0413,E1 24.882,E2 312.7139} C_DIS
LIN {X -76.0881,Y 66.2408,Z 99,A 134.6502,B 24.9222,C -2.0372,E1 24.8783,E2 310.7291} C_DIS
LIN {X -78.0437,Y 63.9271,Z 99,A 136.4203,B 24.9224,C -2.0344,E1 24.8752,E2 308.9575} C_DIS
LIN {X -80.1722,Y 61.2359,Z 99,A 138.1126,B 24.9235,C -2.0204,E1 24.8723,E2 307.2906} C_DIS
LIN {X -81.7506,Y 59.1127,Z 99,A 140.216,B 24.9222,C -2.0371,E1 24.8688,E2 305.1373} C_DIS
LIN {X -85.1866,Y 54.044,Z 99,A 143.3841,B 24.9237,C -2.0166,E1 24.864,E2 302.002} C_DIS
LIN {X -86.6069,Y 51.7367,Z 99,A 145.5056,B 24.9225,C -2.0324,E1 24.8609,E2 299.832} C_DIS
LIN {X -88.6254,Y 48.1952,Z 99,A 147.2161,B 24.9246,C -2.0047,E1 24.8586,E2 298.1785} C_DIS
LIN {X -90.2342,Y 45.1125,Z 99,A 149.1677,B 24.9251,C -1.9981,E1 24.8562,E2 296.2323} C_DIS
LIN {X -92.259,Y 40.8141,Z 99,A 151.7434,B 24.9261,C -1.9857,E1 24.8532,E2 293.6719} C_DIS
LIN {X -93.4072,Y 38.1095,Z 99,A 153.5345,B 24.9261,C -1.9849,E1 24.8512,E2 291.873} C_DIS
LIN {X -94.6491,Y 34.913,Z 99,A 155.5628,B 24.9264,C -1.9816,E1 24.8492,E2 289.841} C_DIS
LIN {X -95.7212,Y 31.8565,Z 99,A 157.1819,B 24.9274,C -1.9684,E1 24.8478,E2 288.2443} C_DIS
LIN {X -96.6288,Y 28.9863,Z 99,A 159.1746,B 24.927,C -1.9727,E1 24.8461,E2 286.2299} C_DIS
LIN {X -97.49,Y 25.9435,Z 99,A 161.0392,B 24.9273,C -1.9693,E1 24.8448,E2 284.3624} C_DIS
LIN {X -98.4181,Y 22.1677,Z 99,A 163.149,B 24.9281,C -1.9589,E1 24.8434,E2 282.265} C_DIS
LIN {X -99.0485,Y 19.1475,Z 99,A 164.8012,B 24.9287,C -1.95,E1 24.8425,E2 280.6244} C_DIS
LIN {X -99.5586,Y 16.292,Z 99,A 166.6169,B 24.9287,C -1.9504,E1 24.8417,E2 278.7969} C_DIS
LIN {X -100.0274,Y 13.1063,Z 99,A 168.2256,B 24.9297,C -1.937,E1 24.841,E2 277.2105} C_DIS
LIN {X -100.5437,Y 8.2613,Z 99,A 171.6309,B 24.9287,C -1.9499,E1 24.8401,E2 273.754} C_DIS
LIN {X -100.766,Y 4.8696,Z 99,A 173.2081,B 24.9301,C -1.9316,E1 24.8399,E2 272.2111} C_DIS
LIN {X -100.8555,Y 2.3836,Z 99,A 175.0759,B 24.9292,C -1.9426,E1 24.8399,E2 270.3058} C_DIS
LIN {X -100.8761,Y -1.2646,Z 99,A 176.5846,B 24.9311,C -1.9166,E1 24.8399,E2 268.85} C_DIS
LIN {X -100.7892,Y -4.3316,Z 99,A 178.3772,B 24.9314,C -1.9127,E1 24.8399,E2 267.0558} C_DIS
LIN {X -100.5706,Y -7.9239,Z 99,A -179.5408,B 24.9318,C -1.9075,E1 24.8404,E2 264.9738} C_DIS
LIN {X -100.2226,Y -11.5197,Z 99,A -177.5842,B 24.9325,C -1.8977,E1 24.841,E2 263.0287} C_DIS
LIN {X -99.8585,Y -14.3362,Z 99,A -175.9244,B 24.9327,C -1.8942,E1 24.8416,E2 261.3674} C_DIS
LIN {X -99.3316,Y -17.6214,Z 99,A -173.9693,B 24.933,C -1.8906,E1 24.8425,E2 259.4095} C_DIS
LIN {X -98.6694,Y -21.0195,Z 99,A -171.9337,B 24.9333,C -1.8868,E1 24.8436,E2 257.3708} C_DIS
LIN {X -97.947,Y -24.1594,Z 99,A -170.1708,B 24.9338,C -1.8789,E1 24.8448,E2 255.6165} C_DIS
LIN {X -97.1271,Y -27.2692,Z 99,A -168.457,B 24.9345,C -1.8694,E1 24.846,E2 253.9153} C_DIS
LIN {X -95.601,Y -32.2128,Z 99,A -165.3312,B 24.9347,C -1.8671,E1 24.8487,E2 250.7772} C_DIS
LIN {X -94.4519,Y -35.4424,Z 99,A -163.3227,B 24.9349,C -1.8634,E1 24.8506,E2 248.7659} C_DIS
LIN {X -92.6354,Y -39.9509,Z 99,A -160.5631,B 24.9355,C -1.8554,E1 24.8535,E2 246.0102} C_DIS
LIN {X -91.1684,Y -43.1955,Z 99,A -158.6328,B 24.9361,C -1.8465,E1 24.8558,E2 244.0906} C_DIS
LIN {X -89.6602,Y -46.2429,Z 99,A -156.5548,B 24.9361,C -1.8462,E1 24.8584,E2 242.002} C_DIS
LIN {X -87.916,Y -49.4784,Z 99,A -154.6216,B 24.9369,C -1.8352,E1 24.861,E2 240.0849} C_DIS
LIN {X -85.7952,Y -53.0717,Z 99,A -152.1322,B 24.937,C -1.8331,E1 24.8646,E2 237.5878} C_DIS
LIN {X -83.7162,Y -56.2932,Z 99,A -149.9862,B 24.9375,C -1.8264,E1 24.8679,E2 235.447} C_DIS
LIN {X -82.3842,Y -58.2261,Z 99,A -148.4012,B 24.9371,C -1.8319,E1 24.8704,E2 233.8411} C_DIS
LIN {X -80.1181,Y -61.306,Z 99,A -146.3825,B 24.9378,C -1.8212,E1 24.8738,E2 231.8382} C_DIS
LIN {X -77.938,Y -64.0562,Z 99,A -144.3613,B 24.9381,C -1.8175,E1 24.8773,E2 229.8165} C_DIS
LIN {X -74.9891,Y -67.4828,Z 99,A -141.7907,B 24.9385,C -1.8118,E1 24.8821,E2 227.2479} C_DIS
LIN {X -72.7995,Y -69.8392,Z 99,A -139.9395,B 24.9387,C -1.8086,E1 24.8856,E2 225.3961} C_DIS
LIN {X -70.8465,Y -71.8192,Z 99,A -138.3695,B 24.9389,C -1.805,E1 24.8887,E2 223.8281} C_DIS
LIN {X -68.2298,Y -74.3096,Z 99,A -136.3431,B 24.9393,C -1.7999,E1 24.8929,E2 221.8056} C_DIS
LIN {X -65.4277,Y -76.7883,Z 99,A -134.1992,B 24.9395,C -1.7964,E1 24.8974,E2 219.6615} C_DIS
LIN {X -62.0207,Y -79.5674,Z 99,A -131.6369,B 24.9397,C -1.7942,E1 24.903,E2 217.095} C_DIS
LIN {X -59.1048,Y -81.7568,Z 99,A -129.5955,B 24.94,C -1.7895,E1 24.9076,E2 215.0574} C_DIS
LIN {X -56.6165,Y -83.4973,Z 99,A -127.9356,B 24.9403,C -1.7844,E1 24.9114,E2 213.4042} C_DIS
LIN {X -54.0306,Y -85.1952,Z 99,A -125.8418,B 24.9397,C -1.7939,E1 24.9164,E2 211.281} C_DIS
LIN {X -50.8444,Y -87.1344,Z 99,A -123.6402,B 24.9397,C -1.7939,E1 24.9217,E2 209.0728} C_DIS
LIN {X -46.8453,Y -89.3464,Z 99,A -121.3833,B 24.9407,C -1.778,E1 24.9271,E2 206.8472} C_DIS
LIN {X -43.6049,Y -90.9717,Z 99,A -119.3651,B 24.941,C -1.7741,E1 24.9322,E2 204.8333} C_DIS
LIN {X -40.9246,Y -92.2102,Z 99,A -117.5445,B 24.9408,C -1.7774,E1 24.9369,E2 203.0002} C_DIS
LIN {X -37.3875,Y -93.7,Z 99,A -115.4194,B 24.9411,C -1.7732,E1 24.9423,E2 200.8803} C_DIS
LIN {X -34.1771,Y -94.9175,Z 99,A -113.5294,B 24.9413,C -1.7693,E1 24.9473,E2 198.9959} C_DIS
LIN {X -30.9842,Y -96.0063,Z 99,A -111.7205,B 24.9417,C -1.7638,E1 24.952,E2 197.1967} C_DIS
LIN {X -26.354,Y -97.3791,Z 99,A -108.3063,B 24.9401,C -1.787,E1 24.9614,E2 193.7217} C_DIS
LIN {X -22.7042,Y -98.2942,Z 99,A -106.9105,B 24.9421,C -1.7581,E1 24.965,E2 192.3926} C_DIS
LIN {X -18.6001,Y -99.1539,Z 99,A -104.2405,B 24.9414,C -1.7679,E1 24.9724,E2 189.6964} C_DIS
LIN {X -14.7107,Y -99.8053,Z 99,A -102.0568,B 24.9416,C -1.7652,E1 24.9784,E2 187.5172} C_DIS
LIN {X -11.1939,Y -100.2608,Z 99,A -100.2041,B 24.942,C -1.7588,E1 24.9835,E2 185.6785} C_DIS
LIN {X -8.3182,Y -100.5391,Z 99,A -98.4394,B 24.9417,C -1.7634,E1 24.9884,E2 183.9019} C_DIS
LIN {X -5.1607,Y -100.751,Z 99,A -96.5664,B 24.9415,C -1.7663,E1 24.9937,E2 182.0213} C_DIS
LIN {X -1.5755,Y -100.8703,Z 99,A -94.5374,B 24.9415,C -1.7663,E1 24.9993,E2 179.9922} C_DIS
LIN {X 0.6904,Y -100.8779,Z 99,A -93.4871,B 24.9421,C -1.7577,E1 25.0022,E2 178.9624} C_DIS
Enddeposition()
LIN {X 0.6904,Y -100.8779,Z 99,A -93.4871,B 24.9421,C -1.7577,E1 25.0022,E2 178.9624} C_DIS
Startdeposition()
$VEL.CP = VEL_PRINT
LIN {X 0.0087,Y -99.9972,Z 99,A -94.6981,B 24.9431,C -1.7422,E1 24.9987,E2 180.2101} C_DIS
LIN {X -5.0535,Y -99.8691,Z 99,A -97.5842,B 24.9431,C -1.7424,E1 24.9907,E2 183.0961} C_DIS
LIN {X -11.0286,Y -99.3876,Z 99,A -100.8232,B 24.9426,C -1.7498,E1 24.9817,E2 186.3192} C_DIS
LIN {X -14.3838,Y -98.9563,Z 99,A -102.9753,B 24.9431,C -1.7424,E1 24.9757,E2 188.4906} C_DIS
LIN {X -20.4642,Y -97.88,Z 99,A -106.3036,B 24.9425,C -1.7513,E1 24.9666,E2 191.8012} C_DIS
LIN {X -23.8206,Y -97.1172,Z 99,A -109.3457,B 24.945,C -1.7138,E1 24.9581,E2 194.9365} C_DIS
LIN {X -28.9387,Y -95.7182,Z 99,A -111.5091,B 24.9428,C -1.7473,E1 24.9525,E2 197.024} C_DIS
LIN {X -32.4195,Y -94.5958,Z 99,A -113.8304,B 24.9432,C -1.7408,E1 24.9463,E2 199.365} C_DIS
LIN {X -36.7604,Y -92.9939,Z 99,A -116.2245,B 24.9424,C -1.7525,E1 24.9401,E2 201.7363} C_DIS
LIN {X -39.9802,Y -91.6555,Z 99,A -118.1864,B 24.9422,C -1.7559,E1 24.9351,E2 203.6947} C_DIS
LIN {X -42.8398,Y -90.3558,Z 99,A -120.3036,B 24.9428,C -1.7467,E1 24.9297,E2 205.8392} C_DIS
LIN {X -46.8313,Y -88.3518,Z 99,A -122.5123,B 24.9418,C -1.7624,E1 24.9243,E2 208.0166} C_DIS
LIN {X -50.1892,Y -86.4892,Z 99,A -124.6442,B 24.9414,C -1.7678,E1 24.9191,E2 210.1417} C_DIS
LIN {X -51.9794,Y -85.4242,Z 99,A -125.9357,B 24.9415,C -1.7661,E1 24.916,E2 211.4412} C_DIS
LIN {X -54.5774,Y -83.79,Z 99,A -127.9091,B 24.9419,C -1.7613,E1 24.9113,E2 213.4326} C_DIS
LIN {X -57.5588,Y -81.7709,Z 99,A -130.2194,B 24.9422,C -1.7561,E1 24.906,E2 215.7631} C_DIS
LIN {X -61.2724,Y -79.0248,Z 99,A -132.9484,B 24.9421,C -1.7579,E1 24.8999,E2 218.4976} C_DIS
LIN {X -63.967,Y -76.8595,Z 99,A -134.4381,B 24.9407,C -1.7787,E1 24.8968,E2 219.9436} C_DIS
LIN {X -66.7302,Y -74.4731,Z 99,A -136.5325,B 24.9404,C -1.7827,E1 24.8924,E2 222.0367} C_DIS
LIN {X -70.6188,Y -70.7981,Z 99,A -139.6566,B 24.9402,C -1.787,E1 24.8861,E2 225.1636} C_DIS
LIN {X -72.9155,Y -68.4287,Z 99,A -141.4913,B 24.9397,C -1.793,E1 24.8826,E2 226.9918} C_DIS
LIN {X -76.5038,Y -64.3939,Z 99,A -144.5739,B 24.9392,C -1.8004,E1 24.8769,E2 230.0707} C_DIS
LIN {X -78.452,Y -62.0035,Z 99,A -146.3981,B 24.9391,C -1.8026,E1 24.8737,E2 231.898} C_DIS
LIN {X -81.5623,Y -57.8517,Z 99,A -149.2761,B 24.9384,C -1.8132,E1 24.8689,E2 234.7649} C_DIS
LIN {X -83.0101,Y -55.7549,Z 99,A -151.05,B 24.9389,C -1.8062,E1 24.8661,E2 236.5643} C_DIS
LIN {X -84.8407,Y -52.9264,Z 99,A -153.3178,B 24.9393,C -1.7998,E1 24.8627,E2 238.8587} C_DIS
LIN {X -86.6594,Y -49.8929,Z 99,A -154.6547,B 24.9373,C -1.8285,E1 24.8609,E2 240.1341} C_DIS
LIN {X -88.1508,Y -47.2108,Z 99,A -156.7129,B 24.9377,C -1.8231,E1 24.8581,E2 242.2161} C_DIS
LIN {X -89.8464,Y -43.8988,Z 99,A -158.6524,B 24.9368,C -1.8355,E1 24.8557,E2 244.1364} C_DIS
LIN {X -91.1151,Y -41.1971,Z 99,A -160.5037,B 24.9368,C -1.8356,E1 24.8535,E2 245.9976} C_DIS
LIN {X -93.7415,Y -34.8133,Z 99,A -164.3265,B 24.9357,C -1.8515,E1 24.8496,E2 249.8038} C_DIS
LIN {X -95.7496,Y -28.8328,Z 99,A -167.8908,B 24.9349,C -1.864,E1 24.8465,E2 253.3587} C_DIS
LIN {X -96.5569,Y -25.9984,Z 99,A -169.7737,B 24.9349,C -1.8626,E1 24.845,E2 255.2559} C_DIS
LIN {X -97.3871,Y -22.6922,Z 99,A -171.815,B 24.9348,C -1.8657,E1 24.8437,E2 257.3018} C_DIS
LIN {X -98.1718,Y -19.0119,Z 99,A -173.9633,B 24.9343,C -1.8727,E1 24.8425,E2 259.4462} C_DIS
LIN {X -98.8051,Y -15.3853,Z 99,A -176.0254,B 24.9337,C -1.8808,E1 24.8415,E2 261.501} C_DIS
LIN {X -99.2779,Y -11.9648,Z 99,A -178.098,B 24.9335,C -1.884,E1 24.8408,E2 263.5785} C_DIS
LIN {X -99.6445,Y -8.3838,Z 99,A 179.8321,B 24.933,C -1.8903,E1 24.8402,E2 265.6458} C_DIS
LIN {X -99.871,Y -5.0183,Z 99,A 177.8031,B 24.9328,C -1.8933,E1 24.8399,E2 267.6798} C_DIS
LIN {X -99.9891,Y -1.2804,Z 99,A 175.5627,B 24.9325,C -1.8969,E1 24.8398,E2 269.9251} C_DIS
LIN {X -99.9723,Y 2.1921,Z 99,A 173.9172,B 24.9313,C -1.9147,E1 24.8398,E2 271.538} C_DIS
LIN {X -99.884,Y 4.7473,Z 99,A 172.0574,B 24.9319,C -1.9064,E1 24.8401,E2 273.4289} C_DIS
LIN {X -99.3142,Y 11.6553,Z 99,A 168.7248,B 24.9294,C -1.9404,E1 24.8409,E2 276.7003} C_DIS
LIN {X -98.9798,Y 14.219,Z 99,A 166.3705,B 24.9312,C -1.9162,E1 24.8418,E2 279.1264} C_DIS
LIN {X -98.4709,Y 17.3992,Z 99,A 165.0064,B 24.9296,C -1.938,E1 24.8424,E2 280.4466} C_DIS
LIN {X -97.9159,Y 20.2895,Z 99,A 163.2183,B 24.9294,C -1.94,E1 24.8434,E2 282.2405} C_DIS
LIN {X -97.2125,Y 23.4296,Z 99,A 161.3657,B 24.929,C -1.9456,E1 24.8446,E2 284.0907} C_DIS
LIN {X -96.1858,Y 27.3396,Z 99,A 159.0875,B 24.9284,C -1.9542,E1 24.8462,E2 286.3616} C_DIS
LIN {X -94.5185,Y 32.6441,Z 99,A 155.763,B 24.928,C -1.9595,E1 24.8491,E2 289.6925} C_DIS
LIN {X -93.2973,Y 35.988,Z 99,A 153.6262,B 24.9278,C -1.9625,E1 24.8512,E2 291.834} C_DIS
LIN {X -91.8214,Y 39.5989,Z 99,A 150.9963,B 24.9282,C -1.9563,E1 24.8541,E2 294.4933} C_DIS
LIN {X -90.3117,Y 42.9315,Z 99,A 149.5007,B 24.9263,C -1.9825,E1 24.8558,E2 295.9346} C_DIS
LIN {X -88.9644,Y 45.6564,Z 99,A 147.6202,B 24.9263,C -1.983,E1 24.8582,E2 297.824} C_DIS
LIN {X -86.3639,Y 50.4047,Z 99,A 144.7093,B 24.9251,C -1.9984,E1 24.8621,E2 300.7134} C_DIS
LIN {X -83.837,Y 54.5027,Z 99,A 141.6141,B 24.9254,C -1.995,E1 24.8667,E2 303.8325} C_DIS
LIN {X -81.928,Y 57.3328,Z 99,A 139.2053,B 24.9261,C -1.9853,E1 24.8706,E2 306.2764} C_DIS
LIN {X -79.6171,Y 60.5027,Z 99,A 137.5768,B 24.9241,C -2.012,E1 24.8733,E2 307.849} C_DIS
LIN {X -77.6726,Y 62.9771,Z 99,A 135.7988,B 24.9237,C -2.0176,E1 24.8763,E2 309.6219} C_DIS
LIN {X -74.6698,Y 66.5103,Z 99,A 132.8181,B 24.924,C -2.0135,E1 24.8818,E2 312.6259} C_DIS
LIN {X -72.1092,Y 69.2779,Z 99,A 130.9343,B 24.9229,C -2.0282,E1 24.8854,E2 314.483} C_DIS
LIN {X -70.0022,Y 71.4071,Z 99,A 129.069,B 24.9229,C -2.0273,E1 24.8891,E2 316.3583} C_DIS
LIN {X -66.8101,Y 74.4015,Z 99,A 126.3694,B 24.9229,C -2.0266,E1 24.8947,E2 319.0704} C_DIS
LIN {X -63.8375,Y 76.9671,Z 99,A 124.3975,B 24.9219,C -2.0411,E1 24.8988,E2 321.0155} C_DIS
LIN {X -60.8835,Y 79.3246,Z 99,A 122.276,B 24.9214,C -2.0472,E1 24.9035,E2 323.1301} C_DIS
LIN {X -57.7606,Y 81.6272,Z 99,A 119.3206,B 24.923,C -2.0268,E1 24.9103,E2 326.1444} C_DIS
LIN {X -54.39,Y 83.9111,Z 99,A 117.6454,B 24.9209,C -2.0537,E1 24.9141,E2 327.7611} C_DIS
LIN {X -49.2036,Y 87.0541,Z 99,A 113.8041,B 24.9214,C -2.0474,E1 24.9234,E2 331.629} C_DIS
LIN {X -46.2436,Y 88.6614,Z 99,A 112.0977,B 24.9206,C -2.0583,E1 24.9276,E2 333.3142} C_DIS
LIN {X -41.1393,Y 91.1412,Z 99,A 108.9627,B 24.9198,C -2.0674,E1 24.9354,E2 336.4354} C_DIS
LIN {X -38.3284,Y 92.3599,Z 99,A 107.1946,B 24.9197,C -2.0695,E1 24.94,E2 338.2028} C_DIS
LIN {X -35.0443,Y 93.6547,Z 99,A 105.0696,B 24.9197,C -2.0686,E1 24.9455,E2 340.3343} C_DIS
LIN {X -31.438,Y 94.9268,Z 99,A 102.5251,B 24.9205,C -2.059,E1 24.9523,E2 342.9066} C_DIS
LIN {X -27.1564,Y 96.2377,Z 99,A 100.3402,B 24.9192,C -2.0751,E1 24.9581,E2 345.0567} C_DIS
LIN {X -23.7605,Y 97.1318,Z 99,A 98.2244,B 24.9194,C -2.0735,E1 24.9638,E2 347.1795} C_DIS
LIN {X -16.2362,Y 98.6691,Z 99,A 94.018,B 24.9186,C -2.0839,E1 24.9753,E2 351.3658} C_DIS
LIN {X -9.6349,Y 99.5315,Z 99,A 89.2303,B 24.9211,C -2.0515,E1 24.9888,E2 356.2335} C_DIS
LIN {X -4.6384,Y 99.8887,Z 99,A 87.5024,B 24.9178,C -2.0934,E1 24.9933,E2 357.8626} C_DIS
LIN {X -2.196,Y 99.9723,Z 99,A 85.1241,B 24.9205,C -2.0586,E1 25.0002,E2 360.3236} C_DIS
LIN {X 2.196,Y 99.9723,Z 99,A 83.1008,B 24.9191,C -2.0766,E1 25.0057,E2 362.3038} C_DIS
LIN {X 7.4565,Y 99.7187,Z 99,A 80.4769,B 24.918,C -2.091,E1 25.013,E2 364.8927} C_DIS
LIN {X 10.9191,Y 99.3981,Z 99,A 78.18,B 24.9189,C -2.0796,E1 25.0194,E2 367.2151} C_DIS
LIN {X 14.9622,Y 98.8703,Z 99,A 75.8728,B 24.9189,C -2.0801,E1 25.0258,E2 369.5192} C_DIS
LIN {X 18.8295,Y 98.2069,Z 99,A 73.5015,B 24.9193,C -2.0747,E1 25.0323,E2 371.9005} C_DIS
LIN {X 24.0368,Y 97.0644,Z 99,A 70.5202,B 24.9192,C -2.0758,E1 25.0404,E2 374.8751} C_DIS
LIN {X 27.4277,Y 96.1608,Z 99,A 68.7395,B 24.9186,C -2.083,E1 25.0451,E2 376.636} C_DIS
LIN {X 31.6191,Y 94.8657,Z 99,A 66.3356,B 24.9185,C -2.0851,E1 25.0515,E2 379.0304} C_DIS
LIN {X 34.4215,Y 93.8847,Z 99,A 64.4913,B 24.919,C -2.0782,E1 25.0564,E2 380.8872} C_DIS
LIN {X 37.8722,Y 92.5466,Z 99,A 62.447,B 24.919,C -2.079,E1 25.0617,E2 382.9252} C_DIS
LIN {X 40.307,Y 91.513,Z 99,A 60.6352,B 24.9199,C -2.0662,E1 25.0664,E2 384.7629} C_DIS
LIN {X 43.1611,Y 90.2014,Z 99,A 59.0388,B 24.9195,C -2.0717,E1 25.0704,E2 386.3421} C_DIS
LIN {X 46.9058,Y 88.3126,Z 99,A 55.9725,B 24.9217,C -2.0436,E1 25.0781,E2 389.4663} C_DIS
LIN {X 50.5986,Y 86.2499,Z 99,A 54.3747,B 24.9195,C -2.0713,E1 25.0818,E2 390.9939} C_DIS
LIN {X 53.7404,Y 84.328,Z 99,A 52.074,B 24.9204,C -2.0608,E1 25.0873,E2 393.312} C_DIS
LIN {X 56.9679,Y 82.1817,Z 99,A 49.9472,B 24.9204,C -2.0608,E1 25.0922,E2 395.4318} C_DIS
LIN {X 60.7654,Y 79.4155,Z 99,A 47.1338,B 24.9211,C -2.0513,E1 25.0986,E2 398.2573} C_DIS
LIN {X 63.5199,Y 77.231,Z 99,A 45.1711,B 24.9212,C -2.0496,E1 25.1028,E2 400.2168} C_DIS
LIN {X 66.0362,Y 75.0899,Z 99,A 43.1624,B 24.9219,C -2.0414,E1 25.1071,E2 402.2368} C_DIS
LIN {X 68.728,Y 72.634,Z 99,A 41.3249,B 24.9214,C -2.0468,E1 25.1108,E2 404.0542} C_DIS
LIN {X 71.1504,Y 70.2621,Z 99,A 39.3668,B 24.9218,C -2.0421,E1 25.1147,E2 406.0151} C_DIS
LIN {X 73.951,Y 67.3094,Z 99,A 36.7782,B 24.923,C -2.0269,E1 25.1196,E2 408.6282} C_DIS
LIN {X 76.6514,Y 64.2174,Z 99,A 34.6645,B 24.9227,C -2.0308,E1 25.1234,E2 410.7232} C_DIS
LIN {X 78.7795,Y 61.5891,Z 99,A 32.6478,B 24.9233,C -2.023,E1 25.127,E2 412.7488} C_DIS
LIN {X 80.8456,Y 58.8491,Z 99,A 30.6444,B 24.9237,C -2.0167,E1 25.1303,E2 414.7574} C_DIS
LIN {X 82.8469,Y 55.9959,Z 99,A 28.8453,B 24.9235,C -2.0194,E1 25.1331,E2 416.5413} C_DIS
LIN {X 85.1643,Y 52.4071,Z 99,A 26.39,B 24.924,C -2.0127,E1 25.1368,E2 419.0001} C_DIS
LIN {X 86.7384,Y 49.7554,Z 99,A 24.5693,B 24.9246,C -2.0059,E1 25.1394,E2 420.8274} C_DIS
LIN {X 88.5706,Y 46.416,Z 99,A 22.5091,B 24.9246,C -2.0047,E1 25.1421,E2 422.8795} C_DIS
LIN {X 90.5049,Y 42.5223,Z 99,A 19.7306,B 24.926,C -1.9864,E1 25.1455,E2 425.6865} C_DIS
LIN {X 92.7277,Y 37.4273,Z 99,A 17.0337,B 24.9253,C -1.9966,E1 25.1484,E2 428.3446} C_DIS
LIN {X 93.5571,Y 35.3019,Z 99,A 15.4823,B 24.9263,C -1.983,E1 25.15,E2 429.9193} C_DIS
LIN {X 95.011,Y 31.1806,Z 99,A 12.9749,B 24.9268,C -1.9754,E1 25.1523,E2 432.4306} C_DIS
LIN {X 96.037,Y 27.8641,Z 99,A 10.95,B 24.9274,C -1.968,E1 25.1539,E2 434.4615} C_DIS
LIN {X 97.4743,Y 22.3147,Z 99,A 7.8704,B 24.9275,C -1.9661,E1 25.156,E2 437.5278} C_DIS
LIN {X 98.0077,Y 19.8424,Z 99,A 6.0772,B 24.9289,C -1.9478,E1 25.157,E2 439.3536} C_DIS
LIN {X 98.8218,Y 15.2775,Z 99,A 3.5296,B 24.9292,C -1.9438,E1 25.1582,E2 441.8956} C_DIS
LIN {X 99.5229,Y 9.7276,Z 99,A -0.5314,B 24.9323,C -1.8997,E1 25.1594,E2 446.0367} C_DIS
LIN {X 99.9096,Y 4.153,Z 99,A -2.5498,B 24.9297,C -1.9365,E1 25.1597,E2 447.9563} C_DIS
LIN {X 99.9928,Y -0.7972,Z 99,A -5.4679,B 24.9306,C -1.9241,E1 25.1597,E2 450.8863} C_DIS
LIN {X 99.9098,Y -4.1464,Z 99,A -7.3949,B 24.9311,C -1.9176,E1 25.1596,E2 452.8172} C_DIS
LIN {X 99.6508,Y -8.306,Z 99,A -10.3147,B 24.9331,C -1.8886,E1 25.159,E2 455.788} C_DIS
LIN {X 99.2659,Y -12.0677,Z 99,A -11.7297,B 24.9315,C -1.9117,E1 25.1585,E2 457.1402} C_DIS
LIN {X 98.1769,Y -18.9854,Z 99,A -16.8657,B 24.9356,C -1.854,E1 25.1561,E2 462.3822} C_DIS
LIN {X 97.0101,Y -24.2595,Z 99,A -18.8544,B 24.9332,C -1.8882,E1 25.1548,E2 464.2788} C_DIS
LIN {X 96.2834,Y -26.9951,Z 99,A -20.8729,B 24.9346,C -1.8672,E1 25.1533,E2 466.3352} C_DIS
LIN {X 94.8063,Y -31.7953,Z 99,A -23.6712,B 24.9351,C -1.8613,E1 25.1509,E2 469.1315} C_DIS
LIN {X 93.7416,Y -34.8137,Z 99,A -25.3392,B 24.935,C -1.8622,E1 25.1493,E2 470.788} C_DIS
LIN {X 92.4583,Y -38.0892,Z 99,A -27.3393,B 24.9354,C -1.8567,E1 25.1472,E2 472.7902} C_DIS
LIN {X 90.8411,Y -41.8,Z 99,A -29.429,B 24.9352,C -1.8588,E1 25.1449,E2 474.8634} C_DIS
LIN {X 89.1414,Y -45.3101,Z 99,A -32.0411,B 24.9367,C -1.8371,E1 25.1416,E2 477.5128} C_DIS
LIN {X 87.1191,Y -49.0871,Z 99,A -34.6631,B 24.9377,C -1.8232,E1 25.138,E2 480.1538} C_DIS
LIN {X 85.4718,Y -51.9011,Z 99,A -36.0247,B 24.9367,C -1.838,E1 25.1361,E2 481.4735} C_DIS
LIN {X 83.8585,Y -54.4719,Z 99,A -37.9235,B 24.9375,C -1.8267,E1 25.1332,E2 483.3896} C_DIS
LIN {X 81.2257,Y -58.3235,Z 99,A -40.4526,B 24.9375,C -1.825,E1 25.1292,E2 485.9102} C_DIS
LIN {X 79.2841,Y -60.936,Z 99,A -42.3364,B 24.938,C -1.8192,E1 25.126,E2 487.7987} C_DIS
LIN {X 77.0611,Y -63.7244,Z 99,A -44.3528,B 24.9383,C -1.8149,E1 25.1225,E2 489.816} C_DIS
LIN {X 75.049,Y -66.0829,Z 99,A -46.2177,B 24.9388,C -1.8068,E1 25.1191,E2 491.6916} C_DIS
LIN {X 72.6618,Y -68.6985,Z 99,A -48.1186,B 24.9388,C -1.8068,E1 25.1155,E2 493.5842} C_DIS
LIN {X 70.3437,Y -71.0699,Z 99,A -50.0012,B 24.9391,C -1.8028,E1 25.1117,E2 495.4682} C_DIS
LIN {X 67.8041,Y -73.4971,Z 99,A -52.0341,B 24.9395,C -1.7972,E1 25.1076,E2 497.5059} C_DIS
LIN {X 65.245,Y -75.7793,Z 99,A -54.0688,B 24.94,C -1.7899,E1 25.1033,E2 499.5498} C_DIS
LIN {X 62.5357,Y -78.0303,Z 99,A -56.0797,B 24.9402,C -1.7857,E1 25.099,E2 501.5629} C_DIS
LIN {X 59.62,Y -80.2802,Z 99,A -58.1875,B 24.9405,C -1.7813,E1 25.0943,E2 503.6735} C_DIS
LIN {X 55.1394,Y -83.4195,Z 99,A -61.0673,B 24.9403,C -1.785,E1 25.0877,E2 506.5348} C_DIS
LIN {X 52.4488,Y -85.1389,Z 99,A -63.1955,B 24.9413,C -1.7698,E1 25.0826,E2 508.6921} C_DIS
LIN {X 49.3247,Y -86.9859,Z 99,A -65.1391,B 24.9412,C -1.7713,E1 25.0779,E2 510.6262} C_DIS
LIN {X 46.411,Y -88.5732,Z 99,A -67.2488,B 24.9419,C -1.7601,E1 25.0727,E2 512.7566} C_DIS
LIN {X 42.8623,Y -90.345,Z 99,A -69.41,B 24.9419,C -1.7607,E1 25.0672,E2 514.9107} C_DIS
LIN {X 38.5439,Y -92.2693,Z 99,A -72.0771,B 24.9421,C -1.7582,E1 25.0604,E2 517.5771} C_DIS
LIN {X 34.1004,Y -94.0018,Z 99,A -74.6387,B 24.9419,C -1.7611,E1 25.0538,E2 520.1264} C_DIS
LIN {X 30.8922,Y -95.1043,Z 99,A -76.5723,B 24.942,C -1.759,E1 25.0486,E2 522.0611} C_DIS
LIN {X 26.5139,Y -96.4177,Z 99,A -79.0535,B 24.9419,C -1.7613,E1 25.042,E2 524.5326} C_DIS
LIN {X 24.2416,Y -97.0144,Z 99,A -81.7656,B 24.9453,C -1.7085,E1 25.0344,E2 527.3657} C_DIS
LIN {X 18.2707,Y -98.3141,Z 99,A -83.9593,B 24.9423,C -1.7545,E1 25.0286,E2 529.4479} C_DIS
LIN {X 12.1841,Y -99.2522,Z 99,A -87.4703,B 24.9424,C -1.7527,E1 25.0189,E2 532.9601} C_DIS
LIN {X 7.0146,Y -99.7498,Z 99,A -90.689,B 24.9431,C -1.742,E1 25.0099,E2 536.2021} C_DIS
LIN {X 1.9169,Y -99.9774,Z 99,A -93.5336,B 24.943,C -1.744,E1 25.002,E2 539.0414} C_DIS
LIN {X 1.9169,Y -99.9774,Z 99,A -93.5336,B 24.943,C -1.744,E1 25.002,E2 539.0414} C_DIS
Enddeposition()
LIN {X 0.6756,Y -99.1024,Z 99,A -93.8439,B 24.941,C -1.7743,E1 25.0013,E2 539.2797} C_DIS
Startdeposition()
$VEL.CP = VEL_PRINT
LIN {X 6.135,Y -98.9204,Z 99,A -90.3954,B 24.9402,C -1.7861,E1 25.011,E2 535.8042} C_DIS
LIN {X 8.8444,Y -98.7142,Z 99,A -88.2447,B 24.9387,C -1.8088,E1 25.0171,E2 533.6009} C_DIS
LIN {X 12.0771,Y -98.3722,Z 99,A -86.9068,B 24.94,C -1.7894,E1 25.0207,E2 532.31} C_DIS
LIN {X 18.4724,Y -97.3729,Z 99,A -83.3302,B 24.9402,C -1.7859,E1 25.0306,E2 528.7454} C_DIS
LIN {X 23.5711,Y -96.2655,Z 99,A -80.0279,B 24.9393,C -1.7995,E1 25.0396,E2 525.4152} C_DIS
LIN {X 27.0025,Y -95.3599,Z 99,A -77.8903,B 24.9389,C -1.805,E1 25.0454,E2 523.268} C_DIS
LIN {X 30.5769,Y -94.2746,Z 99,A -75.764,B 24.9389,C -1.8063,E1 25.0511,E2 521.1426} C_DIS
LIN {X 33.8788,Y -93.139,Z 99,A -74.0323,B 24.9394,C -1.7978,E1 25.0556,E2 519.4343} C_DIS
LIN {X 36.5371,Y -92.1292,Z 99,A -72.0897,B 24.9385,C -1.8116,E1 25.0607,E2 517.4634} C_DIS
LIN {X 40.7437,Y -90.3471,Z 99,A -69.5779,B 24.9385,C -1.8106,E1 25.0671,E2 514.9602} C_DIS
LIN {X 44.3828,Y -88.617,Z 99,A -67.0986,B 24.9379,C -1.8201,E1 25.0734,E2 512.4647} C_DIS
LIN {X 47.6618,Y -86.8977,Z 99,A -65.1429,B 24.9381,C -1.8166,E1 25.0782,E2 510.5229} C_DIS
LIN {X 50.2474,Y -85.4276,Z 99,A -63.3156,B 24.9376,C -1.824,E1 25.0826,E2 508.6837} C_DIS
LIN {X 53.6887,Y -83.3079,Z 99,A -60.0011,B 24.9346,C -1.8672,E1 25.0906,E2 505.2779} C_DIS
LIN {X 58.3198,Y -80.1344,Z 99,A -57.7708,B 24.937,C -1.8335,E1 25.0955,E2 503.1349} C_DIS
LIN {X 61.2387,Y -77.9264,Z 99,A -55.714,B 24.9368,C -1.8357,E1 25.1,E2 501.0805} C_DIS
LIN {X 63.9192,Y -75.7442,Z 99,A -53.6662,B 24.9364,C -1.8422,E1 25.1044,E2 499.0254} C_DIS
LIN {X 66.583,Y -73.4144,Z 99,A -51.6123,B 24.936,C -1.8472,E1 25.1087,E2 496.9677} C_DIS
LIN {X 69.0001,Y -71.1457,Z 99,A -49.7345,B 24.9358,C -1.8503,E1 25.1125,E2 495.0904} C_DIS
LIN {X 71.5827,Y -68.5468,Z 99,A -47.607,B 24.9354,C -1.8559,E1 25.1167,E2 492.9588} C_DIS
LIN {X 74.0374,Y -65.8877,Z 99,A -45.5393,B 24.9351,C -1.8602,E1 25.1205,E2 490.89} C_DIS
LIN {X 76.1958,Y -63.3785,Z 99,A -43.7204,B 24.9351,C -1.8614,E1 25.1238,E2 489.0765} C_DIS
LIN {X 78.0901,Y -61.0316,Z 99,A -41.8648,B 24.9344,C -1.8705,E1 25.127,E2 487.2082} C_DIS
LIN {X 80.6783,Y -57.5644,Z 99,A -38.8759,B 24.9325,C -1.8971,E1 25.132,E2 484.1711} C_DIS
LIN {X 82.8853,Y -54.339,Z 99,A -37.1981,B 24.9337,C -1.88,E1 25.1345,E2 482.542} C_DIS
LIN {X 84.5619,Y -51.6914,Z 99,A -34.5357,B 24.9309,C -1.9195,E1 25.1385,E2 479.7998} C_DIS
LIN {X 87.0589,Y -47.3646,Z 99,A -31.7088,B 24.9305,C -1.9255,E1 25.1423,E2 476.9735} C_DIS
LIN {X 89.2691,Y -43.0545,Z 99,A -29.7616,B 24.9324,C -1.8993,E1 25.1446,E2 475.0987} C_DIS
LIN {X 90.6469,Y -40.0755,Z 99,A -28.0484,B 24.9324,C -1.8976,E1 25.1466,E2 473.3987} C_DIS
LIN {X 91.7045,Y -37.5897,Z 99,A -26.2775,B 24.9315,C -1.9108,E1 25.1485,E2 471.6063} C_DIS
LIN {X 93.0615,Y -34.0912,Z 99,A -23.5795,B 24.9295,C -1.939,E1 25.1512,E2 468.857} C_DIS
LIN {X 94.3352,Y -30.3896,Z 99,A -22.0951,B 24.9313,C -1.9145,E1 25.1524,E2 467.4387} C_DIS
LIN {X 94.9922,Y -28.2689,Z 99,A -20.3788,B 24.9297,C -1.9361,E1 25.1538,E2 465.6814} C_DIS
LIN {X 96.2234,Y -23.7436,Z 99,A -17.2148,B 24.9277,C -1.9631,E1 25.156,E2 462.4719} C_DIS
LIN {X 97.2115,Y -19.3107,Z 99,A -15.4817,B 24.9298,C -1.9352,E1 25.1569,E2 460.8147} C_DIS
LIN {X 98.1407,Y -13.8223,Z 99,A -12.1313,B 24.9286,C -1.9509,E1 25.1584,E2 457.447} C_DIS
LIN {X 98.4758,Y -11.1927,Z 99,A -10.0939,B 24.9268,C -1.9763,E1 25.1591,E2 455.3617} C_DIS
LIN {X 98.8266,Y -7.49,Z 99,A -8.8631,B 24.929,C -1.946,E1 25.1594,E2 454.2096} C_DIS
LIN {X 99.047,Y -3.5495,Z 99,A -6.1866,B 24.9273,C -1.9693,E1 25.1597,E2 451.4942} C_DIS
LIN {X 99.0344,Y 3.8699,Z 99,A -2.2062,B 24.9272,C -1.9706,E1 25.1597,E2 447.5344} C_DIS
LIN {X 98.679,Y 9.2249,Z 99,A 1.1386,B 24.9257,C -1.9902,E1 25.159,E2 444.1632} C_DIS
LIN {X 97.9278,Y 15.258,Z 99,A 5.1748,B 24.9233,C -2.0224,E1 25.1574,E2 440.0748} C_DIS
LIN {X 97.2598,Y 19.0599,Z 99,A 6.8316,B 24.9245,C -2.0061,E1 25.1565,E2 438.4661} C_DIS
LIN {X 96.749,Y 21.5039,Z 99,A 8.5427,B 24.9234,C -2.0213,E1 25.1555,E2 436.729} C_DIS
LIN {X 95.6414,Y 25.9882,Z 99,A 10.9715,B 24.9235,C -2.0198,E1 25.1538,E2 434.3178} C_DIS
LIN {X 94.6318,Y 29.4529,Z 99,A 12.9182,B 24.9235,C -2.0205,E1 25.1522,E2 432.3805} C_DIS
LIN {X 92.9941,Y 34.276,Z 99,A 15.9363,B 24.9226,C -2.0322,E1 25.1495,E2 429.3518} C_DIS
LIN {X 92.0783,Y 36.6665,Z 99,A 17.885,B 24.9208,C -2.0553,E1 25.1474,E2 427.3594} C_DIS
LIN {X 90.6929,Y 39.97,Z 99,A 19.2592,B 24.9225,C -2.0334,E1 25.1459,E2 426.0444} C_DIS
LIN {X 88.6358,Y 44.3449,Z 99,A 22.2721,B 24.9212,C -2.0499,E1 25.1423,E2 423.0088} C_DIS
LIN {X 87.3929,Y 46.7488,Z 99,A 23.8323,B 24.9209,C -2.054,E1 25.1402,E2 421.4471} C_DIS
LIN {X 85.833,Y 49.5518,Z 99,A 25.6915,B 24.9205,C -2.0592,E1 25.1376,E2 419.5852} C_DIS
LIN {X 84.4964,Y 51.7991,Z 99,A 27.5683,B 24.919,C -2.0777,E1 25.1349,E2 417.6744} C_DIS
LIN {X 82.6982,Y 54.6229,Z 99,A 28.9311,B 24.9204,C -2.06,E1 25.1328,E2 416.3602} C_DIS
LIN {X 80.2569,Y 58.1525,Z 99,A 31.5265,B 24.9196,C -2.0707,E1 25.1287,E2 413.7521} C_DIS
LIN {X 78.4065,Y 60.6225,Z 99,A 33.4139,B 24.9189,C -2.0791,E1 25.1254,E2 411.8538} C_DIS
LIN {X 76.0827,Y 63.5147,Z 99,A 35.4881,B 24.9188,C -2.0814,E1 25.1218,E2 409.7838} C_DIS
LIN {X 73.8364,Y 66.1122,Z 99,A 37.9432,B 24.9169,C -2.1044,E1 25.1171,E2 407.2853} C_DIS
LIN {X 71.2728,Y 68.8684,Z 99,A 39.5825,B 24.9182,C -2.0881,E1 25.114,E2 405.6916} C_DIS
LIN {X 68.8803,Y 71.2613,Z 99,A 41.5748,B 24.9178,C -2.0936,E1 25.1101,E2 403.6947} C_DIS
LIN {X 64.8717,Y 74.9299,Z 99,A 44.6381,B 24.9175,C -2.0968,E1 25.1037,E2 400.636} C_DIS
LIN {X 62.3486,Y 77.0409,Z 99,A 46.4714,B 24.9175,C -2.0978,E1 25.0998,E2 398.8074} C_DIS
LIN {X 57.5999,Y 80.6529,Z 99,A 49.9502,B 24.9169,C -2.105,E1 25.092,E2 395.3241} C_DIS
LIN {X 53.9595,Y 83.134,Z 99,A 52.3246,B 24.9171,C -2.1025,E1 25.0865,E2 392.9636} C_DIS
LIN {X 50.8962,Y 85.0442,Z 99,A 54.4568,B 24.9167,C -2.1074,E1 25.0814,E2 390.8266} C_DIS
LIN {X 48.5718,Y 86.3909,Z 99,A 56.6378,B 24.9146,C -2.1336,E1 25.076,E2 388.5899} C_DIS
LIN {X 45.3813,Y 88.1095,Z 99,A 58.2396,B 24.9159,C -2.1175,E1 25.0721,E2 387.0307} C_DIS
LIN {X 42.2342,Y 89.6611,Z 99,A 60.1047,B 24.9162,C -2.1138,E1 25.0675,E2 385.1793} C_DIS
LIN {X 38.8979,Y 91.158,Z 99,A 62.4352,B 24.9154,C -2.1243,E1 25.0615,E2 382.8295} C_DIS
LIN {X 35.4696,Y 92.5457,Z 99,A 64.4967,B 24.9154,C -2.1235,E1 25.0561,E2 380.7745} C_DIS
LIN {X 32.5509,Y 93.6117,Z 99,A 66.8764,B 24.9135,C -2.1471,E1 25.0497,E2 378.3437} C_DIS
LIN {X 28.7504,Y 94.8493,Z 99,A 68.7096,B 24.9148,C -2.1309,E1 25.0449,E2 376.5522} C_DIS
LIN {X 25.1206,Y 95.8739,Z 99,A 70.8393,B 24.9148,C -2.1304,E1 25.0392,E2 374.4271} C_DIS
LIN {X 19.4555,Y 97.1821,Z 99,A 74.1495,B 24.9148,C -2.1302,E1 25.0302,E2 371.1219} C_DIS
LIN {X 15.8573,Y 97.8337,Z 99,A 76.6869,B 24.9136,C -2.1466,E1 25.0231,E2 368.548} C_DIS
LIN {X 12.5723,Y 98.3087,Z 99,A 78.7702,B 24.913,C -2.1531,E1 25.0173,E2 366.4509} C_DIS
LIN {X 8.5059,Y 98.7454,Z 99,A 80.5822,B 24.9147,C -2.1329,E1 25.0124,E2 364.6879} C_DIS
LIN {X 1.4571,Y 99.0992,Z 99,A 85.7267,B 24.9115,C -2.1718,E1 24.9978,E2 359.4524} C_DIS
LIN {X -4.4535,Y 99.0093,Z 99,A 88.8734,B 24.9124,C -2.1607,E1 24.9891,E2 356.3314} C_DIS
LIN {X -9.3431,Y 98.6681,Z 99,A 90.6836,B 24.9155,C -2.1221,E1 24.9843,E2 354.6119} C_DIS
LIN {X -14.3799,Y 98.0615,Z 99,A 93.865,B 24.915,C -2.1292,E1 24.9754,E2 351.4112} C_DIS
LIN {X -17.3545,Y 97.5782,Z 99,A 96.2281,B 24.9133,C -2.1503,E1 24.9688,E2 348.9957} C_DIS
LIN {X -21.5949,Y 96.7292,Z 99,A 98.1226,B 24.9152,C -2.1263,E1 24.9638,E2 347.1558} C_DIS
LIN {X -25.0643,Y 95.8884,Z 99,A 100.2023,B 24.9153,C -2.1249,E1 24.9581,E2 345.0766} C_DIS
LIN {X -28.6436,Y 94.881,Z 99,A 102.6734,B 24.9146,C -2.1339,E1 24.9514,E2 342.5798} C_DIS
LIN {X -33.3777,Y 93.3216,Z 99,A 105.2699,B 24.9157,C -2.1203,E1 24.9447,E2 340.0109} C_DIS
LIN {X -36.892,Y 91.9885,Z 99,A 107.3472,B 24.9162,C -2.114,E1 24.9393,E2 337.944} C_DIS
LIN {X -39.3203,Y 90.9761,Z 99,A 109.9193,B 24.9134,C -2.1489,E1 24.9325,E2 335.2826} C_DIS
LIN {X -44.4728,Y 88.5724,Z 99,A 112.2187,B 24.9166,C -2.1088,E1 24.927,E2 333.0727} C_DIS
LIN {X -47.6776,Y 86.8891,Z 99,A 114.6197,B 24.916,C -2.116,E1 24.921,E2 330.6479} C_DIS
LIN {X -53.1428,Y 83.6582,Z 99,A 117.9696,B 24.9174,C -2.0981,E1 24.9131,E2 327.3302} C_DIS
LIN {X -56.6519,Y 81.3217,Z 99,A 120.3342,B 24.918,C -2.0908,E1 24.9076,E2 324.9751} C_DIS
LIN {X -58.5374,Y 79.9751,Z 99,A 122.0324,B 24.9173,C -2.1004,E1 24.9037,E2 323.2479} C_DIS
LIN {X -62.2758,Y 77.0999,Z 99,A 124.456,B 24.9185,C -2.0841,E1 24.8985,E2 320.8542} C_DIS
LIN {X -66.508,Y 73.4821,Z 99,A 128.2365,B 24.9176,C -2.0961,E1 24.8905,E2 317.0303} C_DIS
LIN {X -69.1632,Y 70.9886,Z 99,A 129.8847,B 24.9192,C -2.0754,E1 24.8872,E2 315.4245} C_DIS
LIN {X -71.8511,Y 68.2665,Z 99,A 132.6172,B 24.9183,C -2.0878,E1 24.8819,E2 312.6507} C_DIS
LIN {X -74.3927,Y 65.4867,Z 99,A 134.4042,B 24.9197,C -2.0689,E1 24.8786,E2 310.9006} C_DIS
LIN {X -77.7153,Y 61.5059,Z 99,A 137.1988,B 24.9209,C -2.0542,E1 24.8737,E2 308.1282} C_DIS
LIN {X -80.5469,Y 57.7484,Z 99,A 140.1691,B 24.9208,C -2.0553,E1 24.8688,E2 305.1409} C_DIS
LIN {X -84.3966,Y 51.9633,Z 99,A 144.1157,B 24.9218,C -2.0416,E1 24.8628,E2 301.2071} C_DIS
LIN {X -85.7056,Y 49.7734,Z 99,A 145.688,B 24.9219,C -2.0406,E1 24.8606,E2 299.629} C_DIS
LIN {X -87.5995,Y 46.3574,Z 99,A 147.764,B 24.9229,C -2.0279,E1 24.8579,E2 297.5723} C_DIS
LIN {X -89.1841,Y 43.2314,Z 99,A 149.565,B 24.9239,C -2.0144,E1 24.8556,E2 295.794} C_DIS
LIN {X -90.0646,Y 41.3675,Z 99,A 151.4479,B 24.9224,C -2.0339,E1 24.8534,E2 293.854} C_DIS
LIN {X -92.9275,Y 34.4588,Z 99,A 155.219,B 24.9248,C -2.0022,E1 24.8495,E2 290.1377} C_DIS
LIN {X -94.9262,Y 28.4915,Z 99,A 158.7925,B 24.9259,C -1.9886,E1 24.8464,E2 286.5761} C_DIS
LIN {X -96.1465,Y 24.0568,Z 99,A 161.7841,B 24.9257,C -1.9912,E1 24.8442,E2 283.5608} C_DIS
LIN {X -96.9368,Y 20.6431,Z 99,A 163.7904,B 24.9262,C -1.9841,E1 24.843,E2 281.5596} C_DIS
LIN {X -98.1033,Y 14.0859,Z 99,A 167.6156,B 24.9272,C -1.9709,E1 24.8413,E2 277.7432} C_DIS
LIN {X -98.4686,Y 11.2541,Z 99,A 169.2912,B 24.9275,C -1.9665,E1 24.8407,E2 276.0683} C_DIS
LIN {X -98.9511,Y 5.5982,Z 99,A 172.6055,B 24.9282,C -1.957,E1 24.84,E2 272.7568} C_DIS
LIN {X -99.0894,Y 1.9882,Z 99,A 174.8922,B 24.9282,C -1.9569,E1 24.8398,E2 270.4565} C_DIS
LIN {X -99.0916,Y -1.8684,Z 99,A 177.0101,B 24.929,C -1.946,E1 24.8398,E2 268.3519} C_DIS
LIN {X -98.9435,Y -5.7346,Z 99,A 179.2102,B 24.9296,C -1.9376,E1 24.8401,E2 266.1586} C_DIS
LIN {X -98.6682,Y -9.3427,Z 99,A -178.5962,B 24.9299,C -1.9343,E1 24.8407,E2 263.9595} C_DIS
LIN {X -98.2796,Y -12.7972,Z 99,A -176.6705,B 24.9305,C -1.9251,E1 24.8413,E2 262.0442} C_DIS
LIN {X -97.7863,Y -16.1406,Z 99,A -174.7632,B 24.9311,C -1.9174,E1 24.8421,E2 260.144} C_DIS
LIN {X -97.2059,Y -19.3396,Z 99,A -172.6817,B 24.9311,C -1.9183,E1 24.8432,E2 258.0481} C_DIS
LIN {X -96.4296,Y -22.8983,Z 99,A -170.6424,B 24.9316,C -1.9096,E1 24.8445,E2 256.0176} C_DIS
LIN {X -95.7363,Y -25.6367,Z 99,A -168.6715,B 24.9312,C -1.916,E1 24.8459,E2 254.0198} C_DIS
LIN {X -93.8023,Y -31.9975,Z 99,A -165.0366,B 24.9325,C -1.8974,E1 24.849,E2 250.4085} C_DIS
LIN {X -92.6717,Y -35.1369,Z 99,A -163.0115,B 24.9327,C -1.895,E1 24.851,E2 248.3777} C_DIS
LIN {X -90.995,Y -39.2769,Z 99,A -160.6067,B 24.9336,C -1.8815,E1 24.8535,E2 245.9917} C_DIS
LIN {X -89.5273,Y -42.5171,Z 99,A -158.5373,B 24.934,C -1.8762,E1 24.856,E2 243.9238} C_DIS
Enddeposition()
END
